# B&R Automation Studio project NAEUL004C00R13L518F00 (part 12)

#### Act_EntP0200Disp.st
```iecst
ACTION Act_EntP0200Disp:

	//Access Address
	p_tyC0005Main ACCESS ADR(tyCommon.tyMain);

	p_tyC0007Notif ACCESS ADR(tyCommon.tyNotif);

	p_tyC0008MsgBox ACCESS ADR(tyP0200OpsGen.tyMsgBoxHide);

	p_tyC0009Info ACCESS ADR(tyCommon.tyInfo);

	p_tyC0010RcyMsg ACCESS ADR(tyP0200OpsGen.tyRcyMsgHide);

	p_tyP0200OpsGen ACCESS ADR(tyP0200OpsGen.tyOps);
	p_tyP0200OpsOven ACCESS ADR(tyP0200OpsGen.tyOven);
	p_tyP0200OpsUSCommB ACCESS ADR(tyP0200OpsGen.tyUSCommB);
	p_tyP0200OpsUSAVSMEMA ACCESS ADR(tyP0200OpsGen.tyUSAVSMEMA);
	p_tyP0200OpsUSBVSMEMA ACCESS ADR(tyP0200OpsGen.tyUSBVSMEMA);
	p_tyP0200OpsUSAVSMEMA1 ACCESS ADR(tyP0200OpsGen.tyUSAVSMEMA1);
	p_tyP0200OpsUSBVSMEMA1 ACCESS ADR(tyP0200OpsGen.tyUSBVSMEMA1);
	p_tyP0200OpsBypsInitConv ACCESS ADR(tyP0200OpsGen.tyBypsInitConv);

	//Display
	tyP0200OpsGen.tyOven.tyLyr.uiRtStat.0	:= NOT(p_tyNtParamCurr.bOvenInfoPrep AND p_tyMcParamCurr.bOvenEn);

	//Communication - Upstream A
	IF p_tyMcParamCurr.eUSCommA = McSetCommModHermes THEN
		tyP0200OpsGen.tyOps.tyBitmapUSAComm.usiValueIdx	:= 1;
		tyP0200OpsGen.tyOps.tyBitmapUSAComm1.usiValueIdx	:= 1;

	ELSIF p_tyMcParamCurr.eUSCommA = McSetCommModSMEMA THEN
		tyP0200OpsGen.tyOps.tyBitmapUSAComm.usiValueIdx	:= 0;
		tyP0200OpsGen.tyOps.tyBitmapUSAComm1.usiValueIdx	:= 0;

	END_IF

	//Communication - Upstream B
	IF p_tyMcParamCurr.eUSCommB = McSetCommModHermes THEN
		tyP0200OpsGen.tyUSCommB.tyBitmapUSBComm.usiValueIdx	:= 1;
		tyP0200OpsGen.tyUSCommB.tyBitmapUSBComm1.usiValueIdx	:= 1;

	ELSIF p_tyMcParamCurr.eUSCommB = McSetCommModSMEMA THEN
		tyP0200OpsGen.tyUSCommB.tyBitmapUSBComm.usiValueIdx	:= 0;
		tyP0200OpsGen.tyUSCommB.tyBitmapUSBComm1.usiValueIdx	:= 0;

	END_IF

	//Virtual SMEMA
	IF (p_tyUsrMgmtCurrUsr.eUsrLvl = UsrMgmtLvl1) OR p_tyNtParamCurr.bVSMEMAPrep = FALSE OR p_tyMcParamCurr.bVSMEMAEn = FALSE OR (p_tyMcParamCurr.eUSCommA = McSetCommModHermes AND p_tyMcParamCurr.eUSCommB = McSetCommModHermes) THEN

		tyP0200OpsGen.tyOps.tyHotspotUSAVSMEMA.bValue		:= FALSE;
		tyP0200OpsGen.tyUSCommB.tyHotspotUSBVSMEMA.bValue	:= FALSE;
		tyP0200OpsGen.tyOps.tyHotspotUSAVSMEMA1.bValue		:= FALSE;
		tyP0200OpsGen.tyUSCommB.tyHotspotUSBVSMEMA1.bValue	:= FALSE;

		memset(ADR(tyP0200OpsGen.tyUSAVSMEMA), 0, SIZEOF(tyP0200OpsGen.tyUSAVSMEMA));
		memset(ADR(tyP0200OpsGen.tyUSBVSMEMA), 0, SIZEOF(tyP0200OpsGen.tyUSBVSMEMA));
		memset(ADR(tyP0200OpsGen.tyUSAVSMEMA1), 0, SIZEOF(tyP0200OpsGen.tyUSAVSMEMA1));
		memset(ADR(tyP0200OpsGen.tyUSBVSMEMA1), 0, SIZEOF(tyP0200OpsGen.tyUSBVSMEMA1));

		fUIInRtStatHide(ADR(tyP0200OpsGen.tyOps.tyHotspotUSAVSMEMA.uiRtStat));
		fUIInRtStatHide(ADR(tyP0200OpsGen.tyUSCommB.tyHotspotUSBVSMEMA.uiRtStat));
		fUIInRtStatHide(ADR(tyP0200OpsGen.tyUSAVSMEMA.tyLyr.uiRtStat));
		fUIInRtStatHide(ADR(tyP0200OpsGen.tyUSBVSMEMA.tyLyr.uiRtStat));

		fUIInRtStatHide(ADR(tyP0200OpsGen.tyOps.tyHotspotUSAVSMEMA1.uiRtStat));
		fUIInRtStatHide(ADR(tyP0200OpsGen.tyUSCommB.tyHotspotUSBVSMEMA1.uiRtStat));
		fUIInRtStatHide(ADR(tyP0200OpsGen.tyUSAVSMEMA1.tyLyr.uiRtStat));
		fUIInRtStatHide(ADR(tyP0200OpsGen.tyUSBVSMEMA1.tyLyr.uiRtStat));

		bVSMEMAUSAEn	:= FALSE;
		bVSMEMAUSBEn	:= FALSE;

	ELSE

		//Upstream A
		IF p_tyMcParamCurr.eUSCommA = McSetCommModHermes THEN
			tyP0200OpsGen.tyOps.tyHotspotUSAVSMEMA.bValue	:= FALSE;
			tyP0200OpsGen.tyOps.tyHotspotUSAVSMEMA1.bValue	:= FALSE;

			memset(ADR(tyP0200OpsGen.tyUSAVSMEMA), 0, SIZEOF(tyP0200OpsGen.tyUSAVSMEMA));

			fUIInRtStatHide(ADR(tyP0200OpsGen.tyOps.tyHotspotUSAVSMEMA.uiRtStat));
			fUIInRtStatHide(ADR(tyP0200OpsGen.tyUSAVSMEMA.tyLyr.uiRtStat));

			memset(ADR(tyP0200OpsGen.tyUSAVSMEMA1), 0, SIZEOF(tyP0200OpsGen.tyUSAVSMEMA1));

			fUIInRtStatHide(ADR(tyP0200OpsGen.tyOps.tyHotspotUSAVSMEMA1.uiRtStat));
			fUIInRtStatHide(ADR(tyP0200OpsGen.tyUSAVSMEMA1.tyLyr.uiRtStat));

		ELSIF p_tyMcParamCurr.eUSCommA = McSetCommModSMEMA THEN

			IF p_tyNtParamCurr.bUIConvDirRL = FALSE THEN
				tyP0200OpsGen.tyOps.tyHotspotUSAVSMEMA1.bValue	:= FALSE;
				fUIInRtStatHide(ADR(tyP0200OpsGen.tyUSAVSMEMA1.tyBtnStat.uiRtStat));
				fUIInRtStatHide(ADR(tyP0200OpsGen.tyUSAVSMEMA1.tyBtnDual.uiRtStat));
				fUIInRtStatHide(ADR(tyP0200OpsGen.tyUSAVSMEMA1.tyBtnNom.uiRtStat));

				memset(ADR(tyP0200OpsGen.tyUSAVSMEMA1), 0, SIZEOF(tyP0200OpsGen.tyUSAVSMEMA1));
				fUIInRtStatHide(ADR(tyP0200OpsGen.tyOps.tyHotspotUSAVSMEMA1.uiRtStat));
				fUIInRtStatHide(ADR(tyP0200OpsGen.tyUSAVSMEMA1.tyLyr.uiRtStat));

				fUIInRtStatOff(ADR(tyP0200OpsGen.tyOps.tyHotspotUSAVSMEMA.uiRtStat));
				fUIInRtStatOff(ADR(tyP0200OpsGen.tyOps.tyHotspotUSAVSMEMA1.uiRtStat));
				//Stat & Dual
				IF p_tyMcParamCurr.tyUSCommASMEMA.eSelection = SMEMASelIPC9851Ext THEN
					fUIInRtStatOff(ADR(tyP0200OpsGen.tyUSAVSMEMA.tyBtnStat.uiRtStat));
					fUIInRtStatOff(ADR(tyP0200OpsGen.tyUSAVSMEMA.tyBtnDual.uiRtStat));
				ELSE
					fUIInRtStatHide(ADR(tyP0200OpsGen.tyUSAVSMEMA.tyBtnStat.uiRtStat));
					fUIInRtStatHide(ADR(tyP0200OpsGen.tyUSAVSMEMA.tyBtnDual.uiRtStat));
				END_IF

			ELSE

				tyP0200OpsGen.tyOps.tyHotspotUSAVSMEMA.bValue	:= FALSE;
				fUIInRtStatHide(ADR(tyP0200OpsGen.tyUSAVSMEMA.tyBtnStat.uiRtStat));
				fUIInRtStatHide(ADR(tyP0200OpsGen.tyUSAVSMEMA.tyBtnDual.uiRtStat));
				fUIInRtStatHide(ADR(tyP0200OpsGen.tyUSAVSMEMA.tyBtnNom.uiRtStat));

				memset(ADR(tyP0200OpsGen.tyUSAVSMEMA), 0, SIZEOF(tyP0200OpsGen.tyUSAVSMEMA));
				fUIInRtStatHide(ADR(tyP0200OpsGen.tyOps.tyHotspotUSAVSMEMA.uiRtStat));
				fUIInRtStatHide(ADR(tyP0200OpsGen.tyUSAVSMEMA.tyLyr.uiRtStat));

				fUIInRtStatOff(ADR(tyP0200OpsGen.tyOps.tyHotspotUSAVSMEMA1.uiRtStat));

				//Stat & Dual
				IF p_tyMcParamCurr.tyUSCommASMEMA.eSelection = SMEMASelIPC9851Ext THEN
					fUIInRtStatOff(ADR(tyP0200OpsGen.tyUSAVSMEMA1.tyBtnStat.uiRtStat));
					fUIInRtStatOff(ADR(tyP0200OpsGen.tyUSAVSMEMA1.tyBtnDual.uiRtStat));
				ELSE
					fUIInRtStatHide(ADR(tyP0200OpsGen.tyUSAVSMEMA1.tyBtnStat.uiRtStat));
					fUIInRtStatHide(ADR(tyP0200OpsGen.tyUSAVSMEMA1.tyBtnDual.uiRtStat));
				END_IF

			END_IF

		END_IF

		//Upstream B
		IF p_tyNtParamCurr.bProjLaneBPrep THEN
			IF p_tyMcParamCurr.eUSCommB = McSetCommModHermes THEN
				tyP0200OpsGen.tyUSCommB.tyHotspotUSBVSMEMA.bValue	:= FALSE;
				tyP0200OpsGen.tyUSCommB.tyHotspotUSBVSMEMA1.bValue	:= FALSE;

				memset(ADR(tyP0200OpsGen.tyUSBVSMEMA), 0, SIZEOF(tyP0200OpsGen.tyUSBVSMEMA));

				fUIInRtStatHide(ADR(tyP0200OpsGen.tyUSCommB.tyHotspotUSBVSMEMA.uiRtStat));
				fUIInRtStatHide(ADR(tyP0200OpsGen.tyUSBVSMEMA.tyLyr.uiRtStat));

				memset(ADR(tyP0200OpsGen.tyUSBVSMEMA1), 0, SIZEOF(tyP0200OpsGen.tyUSBVSMEMA1));

				fUIInRtStatHide(ADR(tyP0200OpsGen.tyUSCommB.tyHotspotUSBVSMEMA1.uiRtStat));
				fUIInRtStatHide(ADR(tyP0200OpsGen.tyUSBVSMEMA1.tyLyr.uiRtStat));

			ELSIF p_tyMcParamCurr.eUSCommB = McSetCommModSMEMA THEN

				IF p_tyNtParamCurr.bUIConvDirRL = FALSE THEN
					tyP0200OpsGen.tyUSCommB.tyHotspotUSBVSMEMA1.bValue	:= FALSE;
					fUIInRtStatHide(ADR(tyP0200OpsGen.tyUSBVSMEMA1.tyBtnStat.uiRtStat));
					fUIInRtStatHide(ADR(tyP0200OpsGen.tyUSBVSMEMA1.tyBtnDual.uiRtStat));
					fUIInRtStatHide(ADR(tyP0200OpsGen.tyUSBVSMEMA1.tyBtnNom.uiRtStat));

					memset(ADR(tyP0200OpsGen.tyUSBVSMEMA1), 0, SIZEOF(tyP0200OpsGen.tyUSBVSMEMA1));
					fUIInRtStatHide(ADR(tyP0200OpsGen.tyUSCommB.tyHotspotUSBVSMEMA1.uiRtStat));
					fUIInRtStatHide(ADR(tyP0200OpsGen.tyUSBVSMEMA1.tyLyr.uiRtStat));

					fUIInRtStatOff(ADR(tyP0200OpsGen.tyUSCommB.tyHotspotUSBVSMEMA.uiRtStat));

					//Stat & Dual
					IF p_tyMcParamCurr.tyUSCommBSMEMA.eSelection = SMEMASelIPC9851Ext THEN
						fUIInRtStatOff(ADR(tyP0200OpsGen.tyUSBVSMEMA.tyBtnStat.uiRtStat));
						fUIInRtStatOff(ADR(tyP0200OpsGen.tyUSBVSMEMA.tyBtnDual.uiRtStat));
					ELSE
						fUIInRtStatHide(ADR(tyP0200OpsGen.tyUSBVSMEMA.tyBtnStat.uiRtStat));
						fUIInRtStatHide(ADR(tyP0200OpsGen.tyUSBVSMEMA.tyBtnDual.uiRtStat));
					END_IF

				ELSE
					tyP0200OpsGen.tyUSCommB.tyHotspotUSBVSMEMA.bValue	:= FALSE;
					fUIInRtStatHide(ADR(tyP0200OpsGen.tyUSBVSMEMA.tyBtnStat.uiRtStat));
					fUIInRtStatHide(ADR(tyP0200OpsGen.tyUSBVSMEMA.tyBtnDual.uiRtStat));
					fUIInRtStatHide(ADR(tyP0200OpsGen.tyUSBVSMEMA.tyBtnNom.uiRtStat));

					memset(ADR(tyP0200OpsGen.tyUSBVSMEMA), 0, SIZEOF(tyP0200OpsGen.tyUSBVSMEMA));
					fUIInRtStatHide(ADR(tyP0200OpsGen.tyUSCommB.tyHotspotUSBVSMEMA.uiRtStat));
					fUIInRtStatHide(ADR(tyP0200OpsGen.tyUSBVSMEMA.tyLyr.uiRtStat));

					fUIInRtStatOff(ADR(tyP0200OpsGen.tyUSCommB.tyHotspotUSBVSMEMA1.uiRtStat));

					//Stat & Dual
					IF p_tyMcParamCurr.tyUSCommBSMEMA.eSelection = SMEMASelIPC9851Ext THEN
						fUIInRtStatOff(ADR(tyP0200OpsGen.tyUSBVSMEMA1.tyBtnStat.uiRtStat));
						fUIInRtStatOff(ADR(tyP0200OpsGen.tyUSBVSMEMA1.tyBtnDual.uiRtStat));
					ELSE
						fUIInRtStatHide(ADR(tyP0200OpsGen.tyUSBVSMEMA1.tyBtnStat.uiRtStat));
						fUIInRtStatHide(ADR(tyP0200OpsGen.tyUSBVSMEMA1.tyBtnDual.uiRtStat));
					END_IF

				END_IF

			END_IF

		END_IF

	END_IF

	//General Operations Arrow Dislay

	IF p_tyNtParamCurr.bUIConvDirRL THEN

		tyP0200OpsGen.tyOps.tyBitmapDir1.usiValueIdx	:= 1;	// <<--
		tyP0200OpsGen.tyOps.tyBitmapDir2.usiValueIdx	:= 1;	// <<--
	ELSE

		tyP0200OpsGen.tyOps.tyBitmapDir1.usiValueIdx	:= 0;	// -->>
		tyP0200OpsGen.tyOps.tyBitmapDir2.usiValueIdx	:= 0;	// -->>

	END_IF

	//Disable AIV function
	IF p_tyNtParamCurr.bProjMagConvLane1Prep THEN
		fUIInRtStatHide(ADR(tyP0200OpsGen.tyOps.tyHotspotOpsAIV.uiMaskRtStat));
		IF p_tyMcParamCurr.bAGVComEn = FALSE THEN
			//			fUIInRtStatHide(ADR(tyP0200OpsGen.tyOps.tyHotspotOpsAIV.uiRtStat));
			fUIInRtStatOff(ADR(tyP0200OpsGen.tyOps.tyHotspotAIVGroup1Mask.uiMaskRtStat));
		ELSE
			//			fUIInRtStatOff(ADR(tyP0200OpsGen.tyOps.tyHotspotOpsAIV.uiRtStat));
			fUIInRtStatHide(ADR(tyP0200OpsGen.tyOps.tyHotspotAIVGroup1Mask.uiMaskRtStat));
		END_IF
	ELSE
		fUIInRtStatHide(ADR(tyP0200OpsGen.tyOps.tyHotspotAIVGroup1Mask.uiMaskRtStat));
		IF p_tyMcParamCurr.bAGVComEn = FALSE THEN
			//	fUIInRtStatHide(ADR(tyP0200OpsGen.tyOps.tyHotspotOpsAIV.uiRtStat));
			fUIInRtStatOff(ADR(tyP0200OpsGen.tyOps.tyHotspotOpsAIV.uiMaskRtStat));
		ELSE
			fUIInRtStatHide(ADR(tyP0200OpsGen.tyOps.tyHotspotOpsAIV.uiMaskRtStat));
		END_IF
	END_IF

	//AutoRcp
	IF NOT(p_bMcParamAutoRcpDisable) AND p_tyNtParamCurr.eAutoRcpPrecededBy =  PrecededBySelf THEN
		fUIInRtStatHide(ADR(tyP0200OpsGen.tyOps.tyNumPitch.uiRtStat));
		fUIInRtStatHide(ADR(tyP0200OpsGen.tyOps.tyNumMinSltRange.uiRtStat));
		fUIInRtStatHide(ADR(tyP0200OpsGen.tyOps.tyNumMaxSltRange.uiRtStat));
		fUIInRtStatHide(ADR(tyP0200OpsGen.tyOps.tyNumPitchRToL.uiRtStat));
		fUIInRtStatHide(ADR(tyP0200OpsGen.tyOps.tyNumMinSltRangeRToL.uiRtStat));
		fUIInRtStatHide(ADR(tyP0200OpsGen.tyOps.tyNumMaxSltRangeRToL.uiRtStat));
	ELSE  //PrecededByF1 OR p_bMcParamAutoRcpDisable
		tyP0200OpsGen.tyOps.tyNumPitch.uiRtStat.0 :=  p_tyNtParamCurr.bUIConvDirRL;
		tyP0200OpsGen.tyOps.tyNumMinSltRange.uiRtStat.0 := p_tyNtParamCurr.bUIConvDirRL;
		tyP0200OpsGen.tyOps.tyNumMaxSltRange.uiRtStat.0 := p_tyNtParamCurr.bUIConvDirRL;
		tyP0200OpsGen.tyOps.tyNumPitchRToL.uiRtStat.0 :=  NOT(p_tyNtParamCurr.bUIConvDirRL);
		tyP0200OpsGen.tyOps.tyNumMinSltRangeRToL.uiRtStat.0 := NOT(p_tyNtParamCurr.bUIConvDirRL);
		tyP0200OpsGen.tyOps.tyNumMaxSltRangeRToL.uiRtStat.0 := NOT(p_tyNtParamCurr.bUIConvDirRL);
	END_IF

END_ACTION
```

#### Act_OptP0200ChgPage.st
```iecst
ACTION Act_OptP0200ChgPage:

	IF tyP0200OpsGen.tyOps.tyHotspotOpsTravLifter.bRtCompl = TRUE THEN
		tyP0200OpsGen.tyOps.tyHotspotOpsTravLifter.bRtCompl	:= FALSE;

		eChgPage	:= UIP0201OpsTravLifter;

	ELSIF tyP0200OpsGen.tyOps.tyHotspotOps2Mag1.bRtCompl = TRUE OR tyP0200OpsGen.tyOps.tyHotspotOps3Mag1.bRtCompl = TRUE THEN
		tyP0200OpsGen.tyOps.tyHotspotOps2Mag1.bRtCompl	:= FALSE;
		tyP0200OpsGen.tyOps.tyHotspotOps3Mag1.bRtCompl	:= FALSE;

		eChgPage	:= UIP0202OpsMag1;

	ELSIF tyP0200OpsGen.tyOps.tyHotspotOps2Mag2.bRtCompl = TRUE OR tyP0200OpsGen.tyOps.tyHotspotOps3Mag2.bRtCompl = TRUE THEN
		tyP0200OpsGen.tyOps.tyHotspotOps2Mag2.bRtCompl	:= FALSE;
		tyP0200OpsGen.tyOps.tyHotspotOps3Mag2.bRtCompl	:= FALSE;

		eChgPage	:= UIP0203OpsMag2;

	ELSIF tyP0200OpsGen.tyOps.tyHotspotOps3Mag3.bRtCompl = TRUE THEN
		tyP0200OpsGen.tyOps.tyHotspotOps3Mag3.bRtCompl	:= FALSE;

		eChgPage	:= UIP0204OpsMag3;

	ELSIF tyP0200OpsGen.tyOps.tyHotspotOpsAIV.bRtCompl = TRUE THEN
		tyP0200OpsGen.tyOps.tyHotspotOpsAIV.bRtCompl	:= FALSE;

		eChgPage	:= UIP0205OpsAIV;

	ELSIF tyP0200OpsGen.tyOps.tyHotspotOpsMagLane1.bRtCompl = TRUE THEN
		tyP0200OpsGen.tyOps.tyHotspotOpsMagLane1.bRtCompl	:= FALSE;

		eChgPage	:= UIP0206OpsMagConv1;

	ELSIF tyP0200OpsGen.tyOps.tyHotspotOpsMagLane2.bRtCompl = TRUE THEN
		tyP0200OpsGen.tyOps.tyHotspotOpsMagLane2.bRtCompl	:= FALSE;

		eChgPage	:= UIP0207OpsMagConv2;

	ELSIF tyP0200OpsGen.tyOps.tyHotspotOpsMagInfo.bRtCompl = TRUE THEN
		tyP0200OpsGen.tyOps.tyHotspotOpsMagInfo.bRtCompl	:= FALSE;

		eChgPage	:= UIP0800MagInfo;

	ELSIF tyP0200OpsGen.tyOven.tyHotspotOven.bRtCompl = TRUE THEN
		tyP0200OpsGen.tyOven.tyHotspotOven.bRtCompl	:= FALSE;

		eChgPage	:= UIP0850OvenInfo;

	END_IF

END_ACTION
```

#### Act_OptP0200UpdtDat.st
```iecst
ACTION Act_OptP0200UpdtDat:

	//PCB Status
	IF p_bPshrConvHvBrd = TRUE THEN
		IF p_bPshrConvGdBrd = TRUE THEN
			tyP0200OpsGen.tyOps.tyBitmapPCB.usiValueIdx	:= 1;
		ELSE
			tyP0200OpsGen.tyOps.tyBitmapPCB.usiValueIdx	:= 2;
		END_IF
	ELSE
		tyP0200OpsGen.tyOps.tyBitmapPCB.usiValueIdx	:= 0;
	END_IF

	//Communication - Mask
	IF p_tyNtParamCurr.bUIConvDirRL = FALSE THEN
		fUIInRtStatHide(ADR(tyP0200OpsGen.tyOps.tyBitmapUSAComm1.uiMaskRtStat));
		fUIInRtStatHide(ADR(tyP0200OpsGen.tyUSCommB.tyBitmapUSBComm1.uiMaskRtStat));
		IF p_tyMcParamCurr.eUSCommA = McSetCommModSMEMA THEN
			fUIInRtStatHide(ADR(tyP0200OpsGen.tyOps.tyBitmapUSAComm.uiMaskRtStat));
		ELSIF p_tyMcParamCurr.eUSCommA = McSetCommModHermes THEN
			IF p_bUSHermesAConnected = TRUE THEN
				fUIInRtStatHide(ADR(tyP0200OpsGen.tyOps.tyBitmapUSAComm.uiMaskRtStat));
			ELSE
				fUIInRtStatOff(ADR(tyP0200OpsGen.tyOps.tyBitmapUSAComm.uiMaskRtStat));
			END_IF
		END_IF

		IF p_tyMcParamCurr.eUSCommB = McSetCommModSMEMA THEN
			fUIInRtStatHide(ADR(tyP0200OpsGen.tyUSCommB.tyBitmapUSBComm.uiMaskRtStat));
		ELSIF p_tyMcParamCurr.eUSCommB = McSetCommModHermes THEN
			IF p_bUSHermesBConnected = TRUE THEN
				fUIInRtStatHide(ADR(tyP0200OpsGen.tyUSCommB.tyBitmapUSBComm.uiMaskRtStat));
			ELSE
				fUIInRtStatOff(ADR(tyP0200OpsGen.tyUSCommB.tyBitmapUSBComm.uiMaskRtStat));
			END_IF
		END_IF
	ELSE
		fUIInRtStatHide(ADR(tyP0200OpsGen.tyOps.tyBitmapUSAComm.uiMaskRtStat));
		fUIInRtStatHide(ADR(tyP0200OpsGen.tyUSCommB.tyBitmapUSBComm.uiMaskRtStat));
		IF p_tyMcParamCurr.eUSCommA = McSetCommModSMEMA THEN
			fUIInRtStatHide(ADR(tyP0200OpsGen.tyOps.tyBitmapUSAComm1.uiMaskRtStat));
		ELSIF p_tyMcParamCurr.eUSCommA = McSetCommModHermes THEN
			IF p_bUSHermesAConnected = TRUE THEN
				fUIInRtStatHide(ADR(tyP0200OpsGen.tyOps.tyBitmapUSAComm1.uiMaskRtStat));
			ELSE
				fUIInRtStatOff(ADR(tyP0200OpsGen.tyOps.tyBitmapUSAComm1.uiMaskRtStat));
			END_IF
		END_IF

		IF p_tyMcParamCurr.eUSCommB = McSetCommModSMEMA THEN
			fUIInRtStatHide(ADR(tyP0200OpsGen.tyUSCommB.tyBitmapUSBComm1.uiMaskRtStat));
		ELSIF p_tyMcParamCurr.eUSCommB = McSetCommModHermes THEN
			IF p_bUSHermesBConnected = TRUE THEN
				fUIInRtStatHide(ADR(tyP0200OpsGen.tyUSCommB.tyBitmapUSBComm1.uiMaskRtStat));
			ELSE
				fUIInRtStatOff(ADR(tyP0200OpsGen.tyUSCommB.tyBitmapUSBComm1.uiMaskRtStat));
			END_IF
		END_IF
	END_IF
	//Communication - Signal
	//USB A
	IF p_tyMcParamCurr.eUSCommA = McSetCommModSMEMA THEN
		IF p_tyNtParamCurr.bUIConvDirRL = FALSE THEN

			IF p_bUSSMEMAADSRdy = TRUE THEN
				tyP0200OpsGen.tyOps.tyBitmapUSOut.usiValueIdx	:= 1;
			ELSE
				tyP0200OpsGen.tyOps.tyBitmapUSOut.usiValueIdx	:= 0;
			END_IF
		ELSE
			IF p_bUSSMEMAADSRdy = TRUE THEN
				tyP0200OpsGen.tyOps.tyBitmapUSOut1.usiValueIdx	:= 1;
			ELSE
				tyP0200OpsGen.tyOps.tyBitmapUSOut1.usiValueIdx	:= 0;
			END_IF
		END_IF

	ELSIF p_tyMcParamCurr.eUSCommA = McSetCommModHermes THEN
		IF p_tyNtParamCurr.bUIConvDirRL = FALSE THEN
			IF p_bUSHermesADSRdy = TRUE THEN
				IF p_bUSHermesADSGdRdy = TRUE THEN
					tyP0200OpsGen.tyOps.tyBitmapUSOut.usiValueIdx	:= 1;
				ELSE
					tyP0200OpsGen.tyOps.tyBitmapUSOut.usiValueIdx	:= 2;
				END_IF
			ELSE
				tyP0200OpsGen.tyOps.tyBitmapUSOut.usiValueIdx		:= 0;
			END_IF
		ELSE
			IF p_bUSHermesADSRdy = TRUE THEN
				IF p_bUSHermesADSGdRdy = TRUE THEN
					tyP0200OpsGen.tyOps.tyBitmapUSOut1.usiValueIdx	:= 1;
				ELSE
					tyP0200OpsGen.tyOps.tyBitmapUSOut1.usiValueIdx	:= 2;
				END_IF
			ELSE
				tyP0200OpsGen.tyOps.tyBitmapUSOut1.usiValueIdx		:= 0;
			END_IF
		END_IF

	END_IF

	//UBA A
	IF p_tyMcParamCurr.eUSCommA = McSetCommModSMEMA THEN

	IF p_tyNtParamCurr.bUIConvDirRL = FALSE THEN
		IF p_bUSSMEMAAUSRdy = TRUE THEN
			IF p_bUSSMEMAAUSGdBrdRdy = TRUE THEN
				tyP0200OpsGen.tyOps.tyBitmapUSIn.usiValueIdx	:= 1;
			ELSE
				tyP0200OpsGen.tyOps.tyBitmapUSIn.usiValueIdx	:= 2;
			END_IF
		ELSE
			tyP0200OpsGen.tyOps.tyBitmapUSIn.usiValueIdx		:= 0;
		END_IF
	ELSE
		IF p_bUSSMEMAAUSRdy = TRUE THEN
			IF p_bUSSMEMAAUSGdBrdRdy = TRUE THEN
				tyP0200OpsGen.tyOps.tyBitmapUSIn1.usiValueIdx	:= 1;
			ELSE
				tyP0200OpsGen.tyOps.tyBitmapUSIn1.usiValueIdx	:= 2;
			END_IF
		ELSE
			tyP0200OpsGen.tyOps.tyBitmapUSIn1.usiValueIdx		:= 0;
		END_IF
	END_IF

	ELSIF p_tyMcParamCurr.eUSCommA = McSetCommModHermes THEN

		IF p_tyNtParamCurr.bUIConvDirRL = FALSE THEN
			IF p_bUSHermesAUSRdy = TRUE THEN
				IF p_bUSHermesAUSGdRdy = TRUE THEN
					tyP0200OpsGen.tyOps.tyBitmapUSIn.usiValueIdx	:= 1;
				ELSE
					tyP0200OpsGen.tyOps.tyBitmapUSIn.usiValueIdx	:= 2;
				END_IF
			ELSE
				tyP0200OpsGen.tyOps.tyBitmapUSIn.usiValueIdx		:= 0;
			END_IF
		ELSE
			IF p_bUSHermesAUSRdy = TRUE THEN
				IF p_bUSHermesAUSGdRdy = TRUE THEN
					tyP0200OpsGen.tyOps.tyBitmapUSIn1.usiValueIdx	:= 1;
				ELSE
					tyP0200OpsGen.tyOps.tyBitmapUSIn1.usiValueIdx	:= 2;
				END_IF
			ELSE
				tyP0200OpsGen.tyOps.tyBitmapUSIn1.usiValueIdx		:= 0;
			END_IF
		END_IF

	END_IF

	//USB B
	IF p_tyMcParamCurr.eUSCommB = McSetCommModSMEMA THEN
		IF p_tyNtParamCurr.bUIConvDirRL = FALSE THEN

			IF p_bUSSMEMABDSRdy = TRUE THEN
				tyP0200OpsGen.tyUSCommB.tyBitmapUSOut.usiValueIdx	:= 1;
			ELSE
				tyP0200OpsGen.tyUSCommB.tyBitmapUSOut.usiValueIdx	:= 0;
			END_IF

		ELSE

			IF p_bUSSMEMABDSRdy = TRUE THEN
				tyP0200OpsGen.tyUSCommB.tyBitmapUSOut1.usiValueIdx	:= 1;
			ELSE
				tyP0200OpsGen.tyUSCommB.tyBitmapUSOut1.usiValueIdx	:= 0;
			END_IF

		END_IF

	ELSIF p_tyMcParamCurr.eUSCommB = McSetCommModHermes THEN

		IF p_tyNtParamCurr.bUIConvDirRL THEN
			IF p_bUSHermesBDSRdy = TRUE THEN
				IF p_bUSHermesBDSGdRdy = TRUE THEN
					tyP0200OpsGen.tyUSCommB.tyBitmapUSOut.usiValueIdx	:= 1;
				ELSE
					tyP0200OpsGen.tyUSCommB.tyBitmapUSOut.usiValueIdx	:= 2;
				END_IF
			ELSE
				tyP0200OpsGen.tyUSCommB.tyBitmapUSOut.usiValueIdx		:= 0;
			END_IF
		ELSE
			IF p_bUSHermesBDSRdy = TRUE THEN
				IF p_bUSHermesBDSGdRdy = TRUE THEN
					tyP0200OpsGen.tyUSCommB.tyBitmapUSOut1.usiValueIdx	:= 1;
				ELSE
					tyP0200OpsGen.tyUSCommB.tyBitmapUSOut1.usiValueIdx	:= 2;
				END_IF
			ELSE
				tyP0200OpsGen.tyUSCommB.tyBitmapUSOut1.usiValueIdx		:= 0;
			END_IF
		END_IF

	END_IF

	//UBA B
	IF p_tyMcParamCurr.eUSCommB = McSetCommModSMEMA THEN

		IF p_tyNtParamCurr.bUIConvDirRL = FALSE THEN
			IF p_bUSSMEMABUSRdy = TRUE THEN
				IF p_bUSSMEMABUSGdBrdRdy = TRUE THEN
					tyP0200OpsGen.tyUSCommB.tyBitmapUSIn.usiValueIdx	:= 1;
				ELSE
					tyP0200OpsGen.tyUSCommB.tyBitmapUSIn.usiValueIdx	:= 2;
				END_IF
			ELSE
				tyP0200OpsGen.tyUSCommB.tyBitmapUSIn.usiValueIdx		:= 0;
			END_IF
		ELSE
			IF p_bUSSMEMABUSRdy = TRUE THEN
				IF p_bUSSMEMABUSGdBrdRdy = TRUE THEN
					tyP0200OpsGen.tyUSCommB.tyBitmapUSIn1.usiValueIdx	:= 1;
				ELSE
					tyP0200OpsGen.tyUSCommB.tyBitmapUSIn1.usiValueIdx	:= 2;
				END_IF
			ELSE
				tyP0200OpsGen.tyUSCommB.tyBitmapUSIn1.usiValueIdx		:= 0;
			END_IF
		END_IF

	ELSIF p_tyMcParamCurr.eUSCommB = McSetCommModHermes THEN

		IF p_tyNtParamCurr.bUIConvDirRL = FALSE THEN
			IF p_bUSHermesBUSRdy = TRUE THEN
				IF p_bUSHermesBUSGdRdy = TRUE THEN
					tyP0200OpsGen.tyUSCommB.tyBitmapUSIn.usiValueIdx	:= 1;
				ELSE
					tyP0200OpsGen.tyUSCommB.tyBitmapUSIn.usiValueIdx	:= 2;
				END_IF
			ELSE
				tyP0200OpsGen.tyUSCommB.tyBitmapUSIn.usiValueIdx		:= 0;
			END_IF
		ELSE
			IF p_bUSHermesBUSRdy = TRUE THEN
				IF p_bUSHermesBUSGdRdy = TRUE THEN
					tyP0200OpsGen.tyUSCommB.tyBitmapUSIn1.usiValueIdx	:= 1;
				ELSE
					tyP0200OpsGen.tyUSCommB.tyBitmapUSIn1.usiValueIdx	:= 2;
				END_IF
			ELSE
				tyP0200OpsGen.tyUSCommB.tyBitmapUSIn1.usiValueIdx		:= 0;
			END_IF
		END_IF

	END_IF

	//Alarm
	IF NOT p_bAlarmErr THEN
		memset(ADR(tyUIAlmData.bAlm) , 0 , SIZEOF(tyUIAlmData.bAlm));
	END_IF

	IF NOT p_bAlarmWarning THEN
		memset(ADR(tyUIAlmData.bWarning) , 0 , SIZEOF(tyUIAlmData.bWarning));
	ELSE
		IF p_bUSHermesAConnected OR p_tyMcParamCurr.eUSCommA = McSetCommModSMEMA THEN
			tyUIAlmData.bWarning[3114] := FALSE;
		END_IF
		IF p_bUSHermesBConnected OR p_tyMcParamCurr.eUSCommB = McSetCommModSMEMA THEN
			tyUIAlmData.bWarning[3281] := FALSE;
		END_IF
	END_IF

	FOR i := 1 TO c_uiP0200TableSize DO
		IF p_bStartupUISettingsLoadDone THEN
			IF p_tyAlarmCurrList[i].eSeverity = AlmSeverityError THEN
				tyUIAlmData.bAlm[p_tyAlarmCurrList[i].udiErrorCode] := p_tyAlarmCurrList[i].bAlm;
			ELSIF p_tyAlarmCurrList[i].eSeverity = AlmSeverityWarning THEN
				tyUIAlmData.bWarning[p_tyAlarmCurrList[i].udiErrorCode] := p_tyAlarmCurrList[i].bWarning;
			END_IF
		END_IF
	END_FOR

	//Magazine Info
	IF NOT(p_tyNtParamCurr.bAutoRcpPrep) OR  ( p_tyNtParamCurr.bAutoRcpPrep AND  p_bMcParamAutoRcpDisable) THEN
		tyP0200OpsGen.tyOps.tyNumMinSltRange.diValue	:= p_tyProdRcpCurrRcp2.diMinSltValue;
		tyP0200OpsGen.tyOps.tyNumMaxSltRange.diValue	:= p_tyProdRcpCurrRcp2.diMaxSltValue;
		tyP0200OpsGen.tyOps.tyNumPitch.diValue			:= p_tyProdRcpCurrRcp2.diPitch;
	ELSIF p_tyNtParamCurr.eAutoRcpPrecededBy =  PrecededByF1 THEN
		tyP0200OpsGen.tyOps.tyNumMinSltRange.diValue	:= p_tyProdRcpCurrRcp1.diMinSltValue; //update immediately based on LCS Running Rcp
		tyP0200OpsGen.tyOps.tyNumMaxSltRange.diValue	:= p_tyProdRcpCurrRcp1.diMaxSltValue;
		tyP0200OpsGen.tyOps.tyNumPitch.diValue			:= p_tyProdRcpCurrRcp1.diPitch;
	END_IF

	//Mag1
	IF p_bBuffer1MagPresent = TRUE THEN
		IF (p_tyNtParamCurr.eCustomerReq = Siemens OR p_tyNtParamCurr.eCustomerReq = We_Fabricate)AND p_iOpsMagConvUL1MESAcptCond <= 0 AND p_tyMcParamCurr.bMESEn THEN
			tyP0200OpsGen.tyOps.tyNumMag1AvlQty.diValue	:= 0;
			tyP0200OpsGen.tyOps.tyNumMag1TtlSlt.diValue	:= 0;
		ELSE
			tyP0200OpsGen.tyOps.tyNumMag1AvlQty.diValue		:= p_tyBuffer1BffrStat.diTtlBrdCap - (p_tyBuffer1BffrStat.diTtlBadBrd + p_tyBuffer1BffrStat.diTtlGdBrd);
			tyP0200OpsGen.tyOps.tyNumMag1TtlSlt.diValue		:= p_tyBuffer1BffrStat.diTtlBrdCap;
		END_IF
	ELSE
		tyP0200OpsGen.tyOps.tyNumMag1AvlQty.diValue		:= 0;
		tyP0200OpsGen.tyOps.tyNumMag1TtlSlt.diValue		:= 0;
	END_IF

	//Mag2
	IF p_bBuffer2MagPresent = TRUE THEN
		IF (p_tyNtParamCurr.eCustomerReq = Siemens OR p_tyNtParamCurr.eCustomerReq = We_Fabricate) AND p_iOpsMagConvUL2MESAcptCond <= 0 AND p_tyMcParamCurr.bMESEn THEN
			tyP0200OpsGen.tyOps.tyNumMag2AvlQty.diValue	:= 0;
			tyP0200OpsGen.tyOps.tyNumMag2TtlSlt.diValue		:= 0;
		ELSE
			tyP0200OpsGen.tyOps.tyNumMag2AvlQty.diValue		:= p_tyBuffer2BffrStat.diTtlBrdCap - (p_tyBuffer2BffrStat.diTtlBadBrd + p_tyBuffer2BffrStat.diTtlGdBrd);
			tyP0200OpsGen.tyOps.tyNumMag2TtlSlt.diValue		:= p_tyBuffer2BffrStat.diTtlBrdCap;
		END_IF
	ELSE
		tyP0200OpsGen.tyOps.tyNumMag2AvlQty.diValue		:= 0;
		tyP0200OpsGen.tyOps.tyNumMag2TtlSlt.diValue		:= 0;
	END_IF
	//Mag3
	IF p_bBuffer3MagPresent = TRUE THEN
		IF (p_tyNtParamCurr.eCustomerReq = Siemens OR p_tyNtParamCurr.eCustomerReq = We_Fabricate) AND p_iOpsMagConvUL3MESAcptCond <= 0 AND  p_tyMcParamCurr.bMESEn THEN
			tyP0200OpsGen.tyOps.tyNumMag3AvlQty.diValue		:= 0;
			tyP0200OpsGen.tyOps.tyNumMag3TtlSlt.diValue		:= 0;
		ELSE
			tyP0200OpsGen.tyOps.tyNumMag3AvlQty.diValue		:= p_tyBuffer3BffrStat.diTtlBrdCap - (p_tyBuffer3BffrStat.diTtlBadBrd + p_tyBuffer3BffrStat.diTtlGdBrd);
			tyP0200OpsGen.tyOps.tyNumMag3TtlSlt.diValue		:= p_tyBuffer3BffrStat.diTtlBrdCap;
		END_IF
	ELSE
		tyP0200OpsGen.tyOps.tyNumMag3AvlQty.diValue		:= 0;
		tyP0200OpsGen.tyOps.tyNumMag3TtlSlt.diValue		:= 0;
	END_IF

	//Oven
	tyP0200OpsGen.tyOven.tyBtnCntrA.bValue				:= p_tyDI.bOvenInfeedSigA;
	tyP0200OpsGen.tyOven.tyBtnCntrB.bValue				:= p_tyDI.bOvenInfeedSigB;
	tyP0200OpsGen.tyOven.tyBtnOvenA.bValue				:= p_tyDO.bOvenInfoSigA;
	tyP0200OpsGen.tyOven.tyBtnOvenB.bValue				:= p_tyDO.bOvenInfoSigB;

	//AIV TCP Bitmap
	IF p_tyNtParamCurr.bProjTCPAGVSigPrep THEN
		tyP0200OpsGen.tyOps.tyBitmapAIVTCP.usiValueIdx := BOOL_TO_USINT (p_bTCPConnected);
	END_IF
END_ACTION
```

#### Act_OptP0200VirtualSMEMA.st
```iecst
ACTION Act_OptP0200VSMEMA:

	//Upstream Virtual SMEMA A
	//Enable / Disable
	IF p_tyNtParamCurr.bUIConvDirRL = FALSE THEN
		IF tyP0200OpsGen.tyOps.tyHotspotUSAVSMEMA.bRtCompl = TRUE THEN
			tyP0200OpsGen.tyOps.tyHotspotUSAVSMEMA.bRtCompl	:= FALSE;

			IF tyP0200OpsGen.tyOps.tyHotspotUSAVSMEMA.bValue = TRUE THEN
				bVSMEMAUSAEn	:= TRUE;

				fUIInRtStatOff(ADR(tyP0200OpsGen.tyUSAVSMEMA.tyLyr.uiRtStat));
				fUIInRtStatHide(ADR(tyP0200OpsGen.tyUSAVSMEMA1.tyLyr.uiRtStat));
			ELSE
				tyP0200OpsGen.tyUSAVSMEMA.tyBtnNom.bValue	:= FALSE;
				tyP0200OpsGen.tyUSAVSMEMA.tyBtnStat.bValue	:= FALSE;
				tyP0200OpsGen.tyUSAVSMEMA.tyBtnDual.bValue	:= FALSE;

				bVSMEMAUSAEn	:= FALSE;

				fUIInRtStatHide(ADR(tyP0200OpsGen.tyUSAVSMEMA.tyLyr.uiRtStat));
				fUIInRtStatHide(ADR(tyP0200OpsGen.tyUSAVSMEMA1.tyLyr.uiRtStat));
			END_IF

		END_IF
	ELSE
		IF tyP0200OpsGen.tyOps.tyHotspotUSAVSMEMA1.bRtCompl = TRUE THEN
			tyP0200OpsGen.tyOps.tyHotspotUSAVSMEMA1.bRtCompl	:= FALSE;

			IF tyP0200OpsGen.tyOps.tyHotspotUSAVSMEMA1.bValue = TRUE THEN
				bVSMEMAUSAEn	:= TRUE;

				fUIInRtStatOff(ADR(tyP0200OpsGen.tyUSAVSMEMA1.tyLyr.uiRtStat));
				fUIInRtStatHide(ADR(tyP0200OpsGen.tyUSAVSMEMA.tyLyr.uiRtStat));
			ELSE
				tyP0200OpsGen.tyUSAVSMEMA.tyBtnNom.bValue	:= FALSE;
				tyP0200OpsGen.tyUSAVSMEMA.tyBtnStat.bValue	:= FALSE;
				tyP0200OpsGen.tyUSAVSMEMA.tyBtnDual.bValue	:= FALSE;

				bVSMEMAUSAEn	:= FALSE;

				fUIInRtStatHide(ADR(tyP0200OpsGen.tyUSAVSMEMA.tyLyr.uiRtStat));
				fUIInRtStatHide(ADR(tyP0200OpsGen.tyUSAVSMEMA1.tyLyr.uiRtStat));
			END_IF

		END_IF

	END_IF

	//Control

	IF p_tyNtParamCurr.bUIConvDirRL = FALSE THEN
		IF tyP0200OpsGen.tyUSAVSMEMA.tyBtnDual.bRtCompl = TRUE THEN
			tyP0200OpsGen.tyUSAVSMEMA.tyBtnDual.bRtCompl	:= FALSE;

			IF tyP0200OpsGen.tyUSAVSMEMA.tyBtnDual.bValue = TRUE THEN
				tyP0200OpsGen.tyUSAVSMEMA.tyBtnNom.bValue	:= TRUE;
				tyP0200OpsGen.tyUSAVSMEMA.tyBtnStat.bValue	:= TRUE;
			ELSE
				tyP0200OpsGen.tyUSAVSMEMA.tyBtnNom.bValue	:= FALSE;
				tyP0200OpsGen.tyUSAVSMEMA.tyBtnStat.bValue	:= FALSE;
			END_IF

		ELSIF tyP0200OpsGen.tyUSAVSMEMA.tyBtnNom.bRtCompl = TRUE THEN
			tyP0200OpsGen.tyUSAVSMEMA.tyBtnNom.bRtCompl	:= FALSE;

			IF tyP0200OpsGen.tyUSAVSMEMA.tyBtnNom.bValue = TRUE THEN
				IF tyP0200OpsGen.tyUSAVSMEMA.tyBtnStat.bValue =  TRUE THEN
					tyP0200OpsGen.tyUSAVSMEMA.tyBtnDual.bValue	:= TRUE;
				END_IF
			ELSE
				tyP0200OpsGen.tyUSAVSMEMA.tyBtnDual.bValue	:= FALSE;
			END_IF

		ELSIF tyP0200OpsGen.tyUSAVSMEMA.tyBtnStat.bRtCompl = TRUE THEN
			tyP0200OpsGen.tyUSAVSMEMA.tyBtnStat.bRtCompl	:= FALSE;

			IF tyP0200OpsGen.tyUSAVSMEMA.tyBtnStat.bValue = TRUE THEN
				IF tyP0200OpsGen.tyUSAVSMEMA.tyBtnNom.bValue =  TRUE THEN
					tyP0200OpsGen.tyUSAVSMEMA.tyBtnDual.bValue	:= TRUE;
				END_IF
			ELSE
				tyP0200OpsGen.tyUSAVSMEMA.tyBtnDual.bValue	:= FALSE;
			END_IF

		END_IF
	ELSE
		IF tyP0200OpsGen.tyUSAVSMEMA1.tyBtnDual.bRtCompl = TRUE THEN
			tyP0200OpsGen.tyUSAVSMEMA1.tyBtnDual.bRtCompl	:= FALSE;

			IF tyP0200OpsGen.tyUSAVSMEMA1.tyBtnDual.bValue = TRUE THEN
				tyP0200OpsGen.tyUSAVSMEMA1.tyBtnNom.bValue	:= TRUE;
				tyP0200OpsGen.tyUSAVSMEMA1.tyBtnStat.bValue	:= TRUE;
			ELSE
				tyP0200OpsGen.tyUSAVSMEMA1.tyBtnNom.bValue	:= FALSE;
				tyP0200OpsGen.tyUSAVSMEMA1.tyBtnStat.bValue	:= FALSE;
			END_IF

		ELSIF tyP0200OpsGen.tyUSAVSMEMA1.tyBtnNom.bRtCompl = TRUE THEN
			tyP0200OpsGen.tyUSAVSMEMA1.tyBtnNom.bRtCompl	:= FALSE;

			IF tyP0200OpsGen.tyUSAVSMEMA1.tyBtnNom.bValue = TRUE THEN
				IF tyP0200OpsGen.tyUSAVSMEMA1.tyBtnStat.bValue =  TRUE THEN
					tyP0200OpsGen.tyUSAVSMEMA1.tyBtnDual.bValue	:= TRUE;
				END_IF
			ELSE
				tyP0200OpsGen.tyUSAVSMEMA1.tyBtnDual.bValue	:= FALSE;
			END_IF

		ELSIF tyP0200OpsGen.tyUSAVSMEMA1.tyBtnStat.bRtCompl = TRUE THEN
			tyP0200OpsGen.tyUSAVSMEMA1.tyBtnStat.bRtCompl	:= FALSE;

			IF tyP0200OpsGen.tyUSAVSMEMA1.tyBtnStat.bValue = TRUE THEN
				IF tyP0200OpsGen.tyUSAVSMEMA1.tyBtnNom.bValue =  TRUE THEN
					tyP0200OpsGen.tyUSAVSMEMA1.tyBtnDual.bValue	:= TRUE;
				END_IF
			ELSE
				tyP0200OpsGen.tyUSAVSMEMA1.tyBtnDual.bValue	:= FALSE;
			END_IF

		END_IF
	END_IF

	//Update
	IF p_tyNtParamCurr.bUIConvDirRL = FALSE THEN
		bVSMEMAUBAA		:= tyP0200OpsGen.tyUSAVSMEMA.tyBtnNom.bValue;
		bVSMEMAUBAAStat	:= tyP0200OpsGen.tyUSAVSMEMA.tyBtnStat.bValue;
	ELSE
		bVSMEMAUBAA		:= tyP0200OpsGen.tyUSAVSMEMA1.tyBtnNom.bValue;
		bVSMEMAUBAAStat	:= tyP0200OpsGen.tyUSAVSMEMA1.tyBtnStat.bValue;
	END_IF

	//Upstream Virtual SMEMA B
	//Enable / Disable
	IF p_tyNtParamCurr.bUIConvDirRL = FALSE THEN
		IF tyP0200OpsGen.tyUSCommB.tyHotspotUSBVSMEMA.bRtCompl = TRUE THEN
			tyP0200OpsGen.tyUSCommB.tyHotspotUSBVSMEMA.bRtCompl	:= FALSE;

			IF tyP0200OpsGen.tyUSCommB.tyHotspotUSBVSMEMA.bValue = TRUE THEN
				bVSMEMAUSBEn	:= TRUE;

				fUIInRtStatOff(ADR(tyP0200OpsGen.tyUSBVSMEMA.tyLyr.uiRtStat));
				fUIInRtStatHide(ADR(tyP0200OpsGen.tyUSBVSMEMA1.tyLyr.uiRtStat));
			ELSE
				tyP0200OpsGen.tyUSBVSMEMA.tyBtnNom.bValue	:= FALSE;
				tyP0200OpsGen.tyUSBVSMEMA.tyBtnStat.bValue	:= FALSE;
				tyP0200OpsGen.tyUSBVSMEMA.tyBtnDual.bValue	:= FALSE;

				bVSMEMAUSBEn	:= FALSE;

				fUIInRtStatHide(ADR(tyP0200OpsGen.tyUSBVSMEMA.tyLyr.uiRtStat));
				fUIInRtStatHide(ADR(tyP0200OpsGen.tyUSBVSMEMA1.tyLyr.uiRtStat));
			END_IF

		END_IF

	ELSE
		IF tyP0200OpsGen.tyUSCommB.tyHotspotUSBVSMEMA1.bRtCompl = TRUE THEN
			tyP0200OpsGen.tyUSCommB.tyHotspotUSBVSMEMA1.bRtCompl	:= FALSE;

			IF tyP0200OpsGen.tyUSCommB.tyHotspotUSBVSMEMA1.bValue = TRUE THEN
				bVSMEMAUSBEn	:= TRUE;

				fUIInRtStatOff(ADR(tyP0200OpsGen.tyUSBVSMEMA1.tyLyr.uiRtStat));
				fUIInRtStatHide(ADR(tyP0200OpsGen.tyUSBVSMEMA.tyLyr.uiRtStat));
			ELSE
				tyP0200OpsGen.tyUSBVSMEMA.tyBtnNom.bValue	:= FALSE;
				tyP0200OpsGen.tyUSBVSMEMA.tyBtnStat.bValue	:= FALSE;
				tyP0200OpsGen.tyUSBVSMEMA.tyBtnDual.bValue	:= FALSE;

				bVSMEMAUSBEn	:= FALSE;

				fUIInRtStatHide(ADR(tyP0200OpsGen.tyUSBVSMEMA.tyLyr.uiRtStat));
				fUIInRtStatHide(ADR(tyP0200OpsGen.tyUSBVSMEMA1.tyLyr.uiRtStat));
			END_IF

		END_IF

	END_IF

	//Control

	IF p_tyNtParamCurr.bUIConvDirRL = FALSE THEN

		IF tyP0200OpsGen.tyUSBVSMEMA.tyBtnDual.bRtCompl = TRUE THEN
			tyP0200OpsGen.tyUSBVSMEMA.tyBtnDual.bRtCompl	:= FALSE;

			IF tyP0200OpsGen.tyUSBVSMEMA.tyBtnDual.bValue = TRUE THEN
				tyP0200OpsGen.tyUSBVSMEMA.tyBtnNom.bValue	:= TRUE;
				tyP0200OpsGen.tyUSBVSMEMA.tyBtnStat.bValue	:= TRUE;
			ELSE
				tyP0200OpsGen.tyUSBVSMEMA.tyBtnNom.bValue	:= FALSE;
				tyP0200OpsGen.tyUSBVSMEMA.tyBtnStat.bValue	:= FALSE;
			END_IF

		ELSIF tyP0200OpsGen.tyUSBVSMEMA.tyBtnNom.bRtCompl = TRUE THEN
			tyP0200OpsGen.tyUSBVSMEMA.tyBtnNom.bRtCompl	:= FALSE;

			IF tyP0200OpsGen.tyUSBVSMEMA.tyBtnNom.bValue = TRUE THEN
				IF tyP0200OpsGen.tyUSBVSMEMA.tyBtnStat.bValue =  TRUE THEN
					tyP0200OpsGen.tyUSBVSMEMA.tyBtnDual.bValue	:= TRUE;
				END_IF
			ELSE
				tyP0200OpsGen.tyUSBVSMEMA.tyBtnDual.bValue	:= FALSE;
			END_IF

		ELSIF tyP0200OpsGen.tyUSBVSMEMA.tyBtnStat.bRtCompl = TRUE THEN
			tyP0200OpsGen.tyUSBVSMEMA.tyBtnStat.bRtCompl	:= FALSE;

			IF tyP0200OpsGen.tyUSBVSMEMA.tyBtnStat.bValue = TRUE THEN
				IF tyP0200OpsGen.tyUSBVSMEMA.tyBtnNom.bValue =  TRUE THEN
					tyP0200OpsGen.tyUSBVSMEMA.tyBtnDual.bValue	:= TRUE;
				END_IF
			ELSE
				tyP0200OpsGen.tyUSBVSMEMA.tyBtnDual.bValue	:= FALSE;
			END_IF

		END_IF

	ELSE

		IF tyP0200OpsGen.tyUSBVSMEMA1.tyBtnDual.bRtCompl = TRUE THEN
			tyP0200OpsGen.tyUSBVSMEMA1.tyBtnDual.bRtCompl	:= FALSE;

			IF tyP0200OpsGen.tyUSBVSMEMA1.tyBtnDual.bValue = TRUE THEN
				tyP0200OpsGen.tyUSBVSMEMA1.tyBtnNom.bValue	:= TRUE;
				tyP0200OpsGen.tyUSBVSMEMA1.tyBtnStat.bValue	:= TRUE;
			ELSE
				tyP0200OpsGen.tyUSBVSMEMA1.tyBtnNom.bValue	:= FALSE;
				tyP0200OpsGen.tyUSBVSMEMA1.tyBtnStat.bValue	:= FALSE;
			END_IF

		ELSIF tyP0200OpsGen.tyUSBVSMEMA1.tyBtnNom.bRtCompl = TRUE THEN
			tyP0200OpsGen.tyUSBVSMEMA1.tyBtnNom.bRtCompl	:= FALSE;

			IF tyP0200OpsGen.tyUSBVSMEMA1.tyBtnNom.bValue = TRUE THEN
				IF tyP0200OpsGen.tyUSBVSMEMA1.tyBtnStat.bValue =  TRUE THEN
					tyP0200OpsGen.tyUSBVSMEMA1.tyBtnDual.bValue	:= TRUE;
				END_IF
			ELSE
				tyP0200OpsGen.tyUSBVSMEMA1.tyBtnDual.bValue	:= FALSE;
			END_IF

		ELSIF tyP0200OpsGen.tyUSBVSMEMA1.tyBtnStat.bRtCompl = TRUE THEN
			tyP0200OpsGen.tyUSBVSMEMA1.tyBtnStat.bRtCompl	:= FALSE;

			IF tyP0200OpsGen.tyUSBVSMEMA1.tyBtnStat.bValue = TRUE THEN
				IF tyP0200OpsGen.tyUSBVSMEMA1.tyBtnNom.bValue =  TRUE THEN
					tyP0200OpsGen.tyUSBVSMEMA1.tyBtnDual.bValue	:= TRUE;
				END_IF
			ELSE
				tyP0200OpsGen.tyUSBVSMEMA1.tyBtnDual.bValue	:= FALSE;
			END_IF

		END_IF
	END_IF

	//Update
	IF p_tyNtParamCurr.bUIConvDirRL = FALSE THEN
		bVSMEMAUBAB		:= tyP0200OpsGen.tyUSBVSMEMA.tyBtnNom.bValue;
		bVSMEMAUBABStat	:= tyP0200OpsGen.tyUSBVSMEMA.tyBtnStat.bValue;
	ELSE
		bVSMEMAUBAB		:= tyP0200OpsGen.tyUSBVSMEMA1.tyBtnNom.bValue;
		bVSMEMAUBABStat	:= tyP0200OpsGen.tyUSBVSMEMA1.tyBtnStat.bValue;
	END_IF

END_ACTION
```

#### Act_OptP0200RcyMsg.st
```iecst
ACTION Act_OptP0200RcyMsg:

	//Recovery Message
	FOR i := 1 TO c_uiP0200TableSize DO

		IF tyP0200OpsGen.tyOps.a_tyHotspotRcyMsg[i].bRtCompl = TRUE THEN
			tyP0200OpsGen.tyOps.a_tyHotspotRcyMsg[i].bRtCompl	:= FALSE;

			tyP0200OpsGen.tyRcyMsg.tyTxtMsg.udiValueIdx := p_tyAlarmRcyList[i];

			IF tyP0200OpsGen.tyRcyMsg.tyTxtMsg.udiValueIdx <> 0 THEN
				p_tyC0010RcyMsg ACCESS ADR(tyP0200OpsGen.tyRcyMsg);
			ELSE
				p_tyC0010RcyMsg ACCESS ADR(tyP0200OpsGen.tyRcyMsgHide);
			END_IF

		END_IF

	END_FOR

	//Close Recovery Message
	IF tyP0200OpsGen.tyRcyMsg.tyHotspotClose.bRtCompl = TRUE THEN
		tyP0200OpsGen.tyRcyMsg.tyHotspotClose.bRtCompl	:= FALSE;

		p_tyC0010RcyMsg ACCESS ADR(tyP0200OpsGen.tyRcyMsgHide);
	END_IF

END_ACTION
```

#### Act_EntP0201Disp.st
```iecst
ACTION Act_EntP0201Disp:

	//Access Address
	p_tyC0004Navi ACCESS ADR(tyP0201OpsTravLifter.tyNaviBack);

	p_tyC0005Main ACCESS ADR(tyCommon.tyMain);

	p_tyC0007Notif ACCESS ADR(tyCommon.tyNotif);

	p_tyC0008MsgBox ACCESS ADR(tyP0201OpsTravLifter.tyMsgBoxHide);

	p_tyC0009Info ACCESS ADR(tyCommon.tyInfo);

	p_tyC0011RcpPopUp ACCESS ADR(tyP0201OpsTravLifter.tyRcpPopUp);

	p_tyP0201OpsTravLif ACCESS ADR(tyP0201OpsTravLifter.tyOps);
	p_tyP0201TravLifIOMonitor ACCESS ADR(tyP0201OpsTravLifter.tyIOMonitor);
	p_tyP0201TravLifIOMonitor1 ACCESS ADR (tyP0201OpsTravLifter.tyIOMonitor1);
	p_tyP0201TravLifBypsInitConv ACCESS ADR(tyP0201OpsTravLifter.tyBypsInitConv);
	p_tyP0201Param ACCESS ADR(tyP0201OpsTravLifter.tyParam);

	//Hermes 1.3
	p_tyE0001OpsQueryBoardInfo ACCESS ADR(tyP0201OpsTravLifter.tyQueryBoardInfo);//new for Hermes 1.3
	p_tyE0002OpsCurrWorkOrder ACCESS ADR(tyP0201OpsTravLifter.tyCurrWorkOrderInfo);//new for Hermes 1.3
	p_tyE0003OpsQueryWorkOrder ACCESS ADR(tyP0201OpsTravLifter.tyQueryWorkOrderInfo);//new for Hermes 1.3
	p_tyE0004OpsBarcodeScanner ACCESS ADR(tyP0201OpsTravLifter.tyBarcodeScanner);//new for Hermes 1.3

	//Display
	fUIInRtStatHide(ADR(tyP0201OpsTravLifter.tyIOMonitor.tyLyr.uiRtStat));
	fUIInRtStatHide(ADR(tyP0201OpsTravLifter.tyParam.tyLyr.uiRtStat));

	tyP0201OpsTravLifter.tyOps.tyBtnChgParam.uiRtStat.0	:= NOT(p_tyMcParamCurr.bChgParamEn);

	tyP0201OpsTravLifter.tyParam.tyNumMaxSlt.diValueMax	:= p_tyMagRcpCurrRcp.diTtlSlt;

	//AutoRcp
	IF (p_bMcParamAutoRcpDisable) THEN
		fUIInRtStatOff(ADR(tyP0201OpsTravLifter.tyOps.tyNumPitch.uiRtStat));
		fUIInRtStatOff(ADR(tyP0201OpsTravLifter.tyOps.tyNumMinSltRange.uiRtStat));
		fUIInRtStatOff(ADR(tyP0201OpsTravLifter.tyOps.tyNumMaxSltRange.uiRtStat));
	ELSE
		IF p_tyNtParamCurr.eAutoRcpPrecededBy =  PrecededBySelf THEN
			fUIInRtStatHide(ADR(tyP0201OpsTravLifter.tyOps.tyNumPitch.uiRtStat));
			fUIInRtStatHide(ADR(tyP0201OpsTravLifter.tyOps.tyNumMinSltRange.uiRtStat));
			fUIInRtStatHide(ADR(tyP0201OpsTravLifter.tyOps.tyNumMaxSltRange.uiRtStat));
		ELSIF p_tyNtParamCurr.eAutoRcpPrecededBy =  PrecededByF1 THEN
			fUIInRtStatOff(ADR(tyP0201OpsTravLifter.tyOps.tyNumPitch.uiRtStat));
			fUIInRtStatOff(ADR(tyP0201OpsTravLifter.tyOps.tyNumMinSltRange.uiRtStat));
			fUIInRtStatOff(ADR(tyP0201OpsTravLifter.tyOps.tyNumMaxSltRange.uiRtStat));
		END_IF
	END_IF

END_ACTION
```

#### Act_OptP0201Navi.st
```iecst
ACTION Act_OptP0201Navi:

	IF tyP0201OpsTravLifter.tyNaviBack.tyBtnBack.bRtCompl = TRUE THEN
		tyP0201OpsTravLifter.tyNaviBack.tyBtnBack.bRtCompl	:= FALSE;
		tyP0201OpsTravLifter.tyNaviBack.tyBtnBack.bValue	:= FALSE;

		eChgPage	:= UIP0200OpsGen;

	END_IF

END_ACTION
```

#### Act_OptP0201UpdtDat.st
```iecst
ACTION Act_OptP0201UpdtDat:

	//Status
	fbMcStatUpdtTm(IN := TRUE);
	IF fbMcStatUpdtTm.Q = TRUE THEN
		fbMcStatUpdtTm(IN := FALSE);

		tyP0201OpsTravLifter.tyOps.tyStringMcStat.sValue	:= p_sOpsTravLifULStepTxt;
	END_IF

	//Width
	IF p_tyNtParamCurr.bAWPrep = TRUE AND p_tyMcParamCurr.bAWDis = FALSE THEN
		tyP0201OpsTravLifter.tyOps.tyNumWidth.diValue		:= p_tyMcParamCurr.diWidthAtHmPosInUM - p_diAWOpenActualPos;
		tyP0201OpsTravLifter.tyOps.tyNumWidth2.diValue		:= p_tyMcParamCurr.diWidthAtHmPosInUM - p_diAWOpenActualPos;
	ELSE
		tyP0201OpsTravLifter.tyOps.tyNumWidth.diValue		:= p_tyProdRcpCurrRcp1.diWidthInUM;
		tyP0201OpsTravLifter.tyOps.tyNumWidth2.diValue		:= p_tyProdRcpCurrRcp1.diWidthInUM2;
	END_IF

	//Program Info
	tyP0201OpsTravLifter.tyOps.tyNumMtrPshrExtSpd.diValue	:= p_tyProdRcpCurrRcp1.diMtrPshrExtSpd;
	tyP0201OpsTravLifter.tyOps.tyNumMtrPshrExtTorq.diValue	:= p_tyProdRcpCurrRcp1.diMtrPshrExtTorq;
	tyP0201OpsTravLifter.tyOps.tyNumPshrOffset.diValue		:= p_tyProdRcpCurrRcp1.diPshrOffset;
	IF p_bMcParamAutoRcpDisable OR p_tyNtParamCurr.eAutoRcpPrecededBy =  PrecededByF1 THEN
		tyP0201OpsTravLifter.tyOps.tyTxtMod.usiValueIdx			:= p_tyProdRcpCurrRcp1.usiMcMod;
		tyP0201OpsTravLifter.tyOps.tyStringProdNm.sValue		:= p_tyProdRcpCurrRcp1.sRcpNm;
		tyP0201OpsTravLifter.tyOps.tyBtnToptoBtm.bValue			:= p_tyProdRcpCurrRcp1.bTopToBtm;
		tyP0201OpsTravLifter.tyOps.tyNumMinSltRange.diValue		:= p_tyProdRcpCurrRcp1.diMinSltValue;
		tyP0201OpsTravLifter.tyOps.tyNumMaxSltRange.diValue		:= p_tyProdRcpCurrRcp1.diMaxSltValue;
		tyP0201OpsTravLifter.tyOps.tyNumPitch.diValue			:= p_tyProdRcpCurrRcp1.diPitch;
	ELSE  //FALSE AutoRcp Mode and eAutoRcpPrecededBy = self
		tyP0201OpsTravLifter.tyOps.tyStringProdNm.sValue		:= pa_tyAutoRcpBrdProps[1].sProductTypeId;
		tyP0201OpsTravLifter.tyOps.tyTxtMod.usiValueIdx			:= p_tyProdRcpCurrRcp0.usiMcMod;
		tyP0201OpsTravLifter.tyOps.tyBtnToptoBtm.bValue			:= p_tyProdRcpCurrRcp0.bTopToBtm;
		tyP0201OpsTravLifter.tyOps.tyNumMtrPshrExtSpd.diValue	:= p_tyProdRcpCurrRcp0.diMtrPshrExtSpd;
		tyP0201OpsTravLifter.tyOps.tyNumMtrPshrExtTorq.diValue	:= p_tyProdRcpCurrRcp0.diMtrPshrExtTorq;
		tyP0201OpsTravLifter.tyOps.tyNumPshrOffset.diValue		:= p_tyProdRcpCurrRcp0.diPshrOffset;
	END_IF

	//PCB Status
	IF p_bPshrConvHvBrd = TRUE THEN
		IF p_bPshrConvGdBrd = TRUE THEN
			tyP0201OpsTravLifter.tyOps.tyBitmapPCB.usiValueIdx	:= 1;
		ELSE
			tyP0201OpsTravLifter.tyOps.tyBitmapPCB.usiValueIdx	:= 2;
		END_IF
	ELSE
		tyP0201OpsTravLifter.tyOps.tyBitmapPCB.usiValueIdx	:= 0;
	END_IF

	//Product Recipe 254
	tyP0201OpsTravLifter.tyOps.tyHotspotShowLRcp.uiRtStat.0 := NOT(tyP0201OpsTravLifter.tyOps.tyStringProdNm.sValue <> '');

	IF tyP0201OpsTravLifter.tyOps.tyHotspotShowLRcp.bRtCompl = TRUE THEN
		tyP0201OpsTravLifter.tyOps.tyHotspotShowLRcp.bRtCompl := FALSE;

		fUIInRtStatOff(ADR(tyP0201OpsTravLifter.tyRcpPopUp.tyLyr.uiRtStat));

		tyP0201OpsTravLifter.tyRcpPopUp.tyStringInfo.sValue  := p_tyProdRcpCurrRcp1.sRcpNm;

	ELSIF tyP0201OpsTravLifter.tyRcpPopUp.tyHotspotClose.bRtCompl = TRUE THEN
		tyP0201OpsTravLifter.tyRcpPopUp.tyHotspotClose.bRtCompl := FALSE;

		fUIInRtStatHide(ADR(tyP0201OpsTravLifter.tyRcpPopUp.tyLyr.uiRtStat));
	END_IF

END_ACTION
```

#### Act_OptP0201IOMonitor.st
```iecst
ACTION Act_OptP0201IOMonitor:

	IF tyP0201OpsTravLifter.tyOps.tyHotspotIOMonitor.bRtCompl = TRUE THEN
		tyP0201OpsTravLifter.tyOps.tyHotspotIOMonitor.bRtCompl	:= FALSE;

		fUIInRtStatOff(ADR(tyP0201OpsTravLifter.tyIOMonitor.tyLyr.uiRtStat));

		p_tyC0004Navi ACCESS ADR(tyP0201OpsTravLifter.tyNaviHide);

	ELSIF tyP0201OpsTravLifter.tyIOMonitor.tyHotspotClose.bRtCompl = TRUE THEN
		tyP0201OpsTravLifter.tyIOMonitor.tyHotspotClose.bRtCompl	:= FALSE;
		fUIInRtStatHide(ADR(tyP0201OpsTravLifter.tyIOMonitor.tyLyr.uiRtStat));

		IF bUITravLifShowIOMonitor2 THEN
			fUIInRtStatOff(ADR(tyP0201OpsTravLifter.tyIOMonitor1.tyLyr.uiRtStat));
		ELSE
			p_tyC0004Navi ACCESS ADR(tyP0201OpsTravLifter.tyNaviBack);
		END_IF

	ELSIF tyP0201OpsTravLifter.tyIOMonitor1.tyHotspotClose.bRtCompl = TRUE THEN
		tyP0201OpsTravLifter.tyIOMonitor1.tyHotspotClose.bRtCompl	:= FALSE;

		fUIInRtStatHide(ADR(tyP0201OpsTravLifter.tyIOMonitor1.tyLyr.uiRtStat));

		p_tyC0004Navi ACCESS ADR(tyP0201OpsTravLifter.tyNaviBack);
	END_IF

	IF tyP0201OpsTravLifter.tyIOMonitor.tyLyr.uiRtStat.0 = FALSE THEN

		//Digital Input
		tyP0201OpsTravLifter.tyIOMonitor.tyBtnSafetyRlySig.bValue			:= p_tyDI.bSafetyRlySig;
		tyP0201OpsTravLifter.tyIOMonitor.tyBtnEStop.bValue					:= p_tyDI.bEStopSig;
		tyP0201OpsTravLifter.tyIOMonitor.tyBtnCoverSWSig.bValue				:= p_tyDI.bCoverSWSig;
		tyP0201OpsTravLifter.tyIOMonitor.tyBtnUBAA.bValue					:= p_tyDI.bUBAA;
		tyP0201OpsTravLifter.tyIOMonitor.tyBtnUBAB.bValue					:= p_tyDI.bUBAB;
		tyP0201OpsTravLifter.tyIOMonitor.tyBtnUBAAStat.bValue				:= p_tyDI.bUBAAStat;
		tyP0201OpsTravLifter.tyIOMonitor.tyBtnUBABStat.bValue				:= p_tyDI.bUBABStat;
		tyP0201OpsTravLifter.tyIOMonitor.tyBtnPshrExtRS.bValue				:= p_tyDI.bPusherExtRS;
		tyP0201OpsTravLifter.tyIOMonitor.tyBtnPshrRetRS.bValue				:= p_tyDI.bPusherRetRS;
		tyP0201OpsTravLifter.tyIOMonitor.tyBtnConvLftSen.bValue				:= p_tyDI.bConvLftSen;
		tyP0201OpsTravLifter.tyIOMonitor.tyBtnConvMidSen.bValue				:= p_tyDI.bConvMidSen;
		tyP0201OpsTravLifter.tyIOMonitor.tyBtnConvRgtSen.bValue				:= p_tyDI.bConvRgtSen;
		tyP0201OpsTravLifter.tyIOMonitor.tyBtnConvClrSen.bValue				:= p_tyDI.bConvClrSen;
		tyP0201OpsTravLifter.tyIOMonitor.tyBtnOvenInfeedSigA.bValue			:= p_tyDI.bOvenInfeedSigA;
		tyP0201OpsTravLifter.tyIOMonitor.tyBtnOvenInfeedSigB.bValue			:= p_tyDI.bOvenInfeedSigB;
		tyP0201OpsTravLifter.tyIOMonitor.tyBtnLifterTmBeltSen.bValue		:= p_tyDI.bLifterTimingBeltSen;
		tyP0201OpsTravLifter.tyIOMonitor.tyBtnInletShutterOpenSen.bValue	:= p_tyDI.bInShutterOpenRS;
		tyP0201OpsTravLifter.tyIOMonitor.tyBtnInletShutterCloseSen.bValue	:= p_tyDI.bInShutterCloseRS;
		tyP0201OpsTravLifter.tyIOMonitor.tyBtnOutletShutterOpenSen.bValue	:= p_tyDI.bOutShutterOpenRS;
		tyP0201OpsTravLifter.tyIOMonitor.tyBtnOutletShutterCloseSen.bValue	:= p_tyDI.bOutShutterCloseRS;
		tyP0201OpsTravLifter.tyIOMonitor.tyBtnOutletShutterOpenSen2.bValue	:= p_tyDI.bOutShutterOpenRS2;
		tyP0201OpsTravLifter.tyIOMonitor.tyBtnOutletShutterCloseSen2.bValue	:= p_tyDI.bOutShutterCloseRS2;
		tyP0201OpsTravLifter.tyIOMonitor.tyBtnOutletShutterOpenSen3.bValue	:= p_tyDI.bOutShutterOpenRS3;
		tyP0201OpsTravLifter.tyIOMonitor.tyBtnOutletShutterCloseSen3.bValue	:= p_tyDI.bOutShutterCloseRS3;
		tyP0201OpsTravLifter.tyIOMonitor.tyBtnAntiJamSen.bValue				:= p_tyDI.bPshrAntiJam;
		tyP0201OpsTravLifter.tyIOMonitor.tyBtnInletStopperASensor.bValue	:= p_tyDI.bInletStopperASen;

		//Digital Output
		tyP0201OpsTravLifter.tyIOMonitor.tyBtnSafetyRlyRst.bValue			:= p_tyDO.bSafetyRlyRst;
		tyP0201OpsTravLifter.tyIOMonitor.tyBtnTLGreen.bValue				:= p_tyDO.bTLGreen;
		tyP0201OpsTravLifter.tyIOMonitor.tyBtnTLAmber.bValue				:= p_tyDO.bTLAmber;
		tyP0201OpsTravLifter.tyIOMonitor.tyBtnTLRed.bValue					:= p_tyDO.bTLRed;
		tyP0201OpsTravLifter.tyIOMonitor.tyBtnBuzzer.bValue					:= p_tyDO.bBuzzer;
		tyP0201OpsTravLifter.tyIOMonitor.tyBtnUSBA.bValue					:= p_tyDO.bUSBA;
		tyP0201OpsTravLifter.tyIOMonitor.tyBtnUSBB.bValue					:= p_tyDO.bUSBB;
		tyP0201OpsTravLifter.tyIOMonitor.tyBtnOvenInfoSigA.bValue			:= p_tyDO.bOvenInfoSigA;
		tyP0201OpsTravLifter.tyIOMonitor.tyBtnOvenInfoSigB.bValue			:= p_tyDO.bOvenInfoSigB;
		tyP0201OpsTravLifter.tyIOMonitor.tyBtnPshrExtCtrl.bValue			:= p_tyDO.bPusherExtCtrl;
		tyP0201OpsTravLifter.tyIOMonitor.tyBtnStopperUnBlkCtrlA.bValue		:= p_tyDO.bStopperUnBlkCtrlA;
		tyP0201OpsTravLifter.tyIOMonitor.tyBtnStopperUnBlkCtrlB.bValue		:= p_tyDO.bStopperUnBlkCtrlB;
		tyP0201OpsTravLifter.tyIOMonitor.tyBtnInShutterOpenCtrl.bValue		:= p_tyDO.bInShutterOpenCtrl;
		tyP0201OpsTravLifter.tyIOMonitor.tyBtnInShutterCloseCtrl.bValue		:= p_tyDO.bInShutterCloseCtrl;
		tyP0201OpsTravLifter.tyIOMonitor.tyBtnOutShutterOpenCtrl.bValue		:= p_tyDO.bOutShutterOpenCtrl;
		tyP0201OpsTravLifter.tyIOMonitor.tyBtnOutShutterCloseCtrl.bValue	:= p_tyDO.bOutShutterCloseCtrl;
		tyP0201OpsTravLifter.tyIOMonitor.tyBtnOutShutterOpenCtrl2.bValue	:= p_tyDO.bOutShutterOpenCtrl2;
		tyP0201OpsTravLifter.tyIOMonitor.tyBtnOutShutterCloseCtrl2.bValue	:= p_tyDO.bOutShutterCloseCtrl2;
		tyP0201OpsTravLifter.tyIOMonitor.tyBtnOutShutterOpenCtrl3.bValue	:= p_tyDO.bOutShutterOpenCtrl3;
		tyP0201OpsTravLifter.tyIOMonitor.tyBtnOutShutterCloseCtrl3.bValue	:= p_tyDO.bOutShutterCloseCtrl3;
		tyP0201OpsTravLifter.tyIOMonitor.tyBtnPshrMtrOn.bValue				:= p_tyDO.bPusherConvMtrOn;

	ELSIF tyP0201OpsTravLifter.tyIOMonitor1.tyLyr.uiRtStat.0 = FALSE THEN
		tyP0201OpsTravLifter.tyIOMonitor1.tyBtnScannerComplSig.bValue		:= p_tyDI.diScanComplSig;
		tyP0201OpsTravLifter.tyIOMonitor1.tyBtnPCBPresentSen.bValue			:= p_tyDI.diPCBScanSen;

		tyP0201OpsTravLifter.tyIOMonitor1.tyBtnTrigScannerSig.bValue		:= p_tyDO.diScanTrigSig;
		tyP0201OpsTravLifter.tyIOMonitor1.tyBtnPCBExitMag1.bValue			:= p_tyDO.diMag1ExitPCB;
		tyP0201OpsTravLifter.tyIOMonitor1.tyBtnPCBExitMag2.bValue			:= p_tyDO.diMag2ExitPCB;
		tyP0201OpsTravLifter.tyIOMonitor1.tyBtnPCBExitMag3.bValue			:= p_tyDO.diMag3ExitPCB;
	END_IF

END_ACTION
```

#### Act_OptP0201ChgParam.st
```iecst
ACTION Act_OptP0201ChgParam:

	tyP0201OpsTravLifter.tyParam.tyNumMinSlt.diValueMax			:= tyP0201OpsTravLifter.tyParam.tyNumMaxSlt.diValue;
	tyP0201OpsTravLifter.tyParam.tyNumMaxSlt.diValueMin			:= tyP0201OpsTravLifter.tyParam.tyNumMinSlt.diValue;
	tyP0201OpsTravLifter.tyParam.tyNumPitch.diValueMax			:= tyP0201OpsTravLifter.tyParam.tyNumMaxSlt.diValue - tyP0201OpsTravLifter.tyParam.tyNumMinSlt.diValue + 1;
	tyP0201OpsTravLifter.tyParam.tyNumPitch.diValueMin			:= 1;
	tyP0201OpsTravLifter.tyOps.tyBtnChgParam.uiRtStat.0			:= NOT(p_tyMcParamCurr.bChgParamEn);

	tyP0201OpsTravLifter.tyParam.tyNumPshrExtSpeed.diValueMin 	:= p_tyNtParamCurr.tyProdRcpMtrPshrExtSpd.diMin;
	tyP0201OpsTravLifter.tyParam.tyNumPshrExtSpeed.diValueMax 	:= p_tyNtParamCurr.tyProdRcpMtrPshrExtSpd.diMax;
	tyP0201OpsTravLifter.tyParam.tyNumPshrExtTorque.diValueMin	:= p_tyNtParamCurr.tyProdRcpMtrPshrExtTorq.diMin;
	tyP0201OpsTravLifter.tyParam.tyNumPshrExtTorque.diValueMax	:= p_tyNtParamCurr.tyProdRcpMtrPshrExtTorq.diMax;
	tyP0201OpsTravLifter.tyParam.tyNumPshrExtSpeed.uiRtStat.0	:= NOT p_tyNtParamCurr.bProjMotorizedPusherPrep;
	tyP0201OpsTravLifter.tyParam.tyNumPshrExtTorque.uiRtStat.0	:= NOT p_tyNtParamCurr.bProjMotorizedPusherPrep;

	IF (tyP0201OpsTravLifter.tyOps.tyNumWidth.diValue) <> 0 THEN
		tyP0201OpsTravLifter.tyParam.tyNumPshrOffset.diValueMin := -(tyP0201OpsTravLifter.tyOps.tyNumWidth.diValue/2 - p_tyMcParamCurr.diAWPusherAtHmPosInUM - IPshrSafeDistanceValue);
		tyP0201OpsTravLifter.tyParam.tyNumPshrOffset.diValueMax := (tyP0201OpsTravLifter.tyOps.tyNumWidth.diValue/2 - p_tyMcParamCurr.diAWPusherAtHmPosInUM - IPshrSafeDistanceValue);
	ELSE
		tyP0201OpsTravLifter.tyParam.tyNumPshrOffset.diValueMin := 0;
		tyP0201OpsTravLifter.tyParam.tyNumPshrOffset.diValueMax := 0;
	END_IF

	//Control
	IF tyP0201OpsTravLifter.tyOps.tyBtnChgParam.bRtCompl = TRUE THEN
		tyP0201OpsTravLifter.tyOps.tyBtnChgParam.bRtCompl	:= FALSE;

		tyProdRcpCurrRcpWr	:= p_tyProdRcpCurrRcp0;

		tyP0201OpsTravLifter.tyParam.tyDrpDnMcMode.usiValueIdx	:= p_tyProdRcpCurrRcp0.usiMcMod;
		tyP0201OpsTravLifter.tyParam.tyNumMinSlt.diValue		:= p_tyProdRcpCurrRcp0.diMinSltValue;
		tyP0201OpsTravLifter.tyParam.tyNumMaxSlt.diValue		:= p_tyProdRcpCurrRcp0.diMaxSltValue;
		tyP0201OpsTravLifter.tyParam.tyNumPitch.diValue			:= p_tyProdRcpCurrRcp0.diPitch;
		tyP0201OpsTravLifter.tyParam.tyBtnToptoBtm.bValue		:= p_tyProdRcpCurrRcp0.bTopToBtm;
		tyP0201OpsTravLifter.tyParam.tyNumPshrExtSpeed.diValue 	:= p_tyProdRcpCurrRcp0.diMtrPshrExtSpd;
		tyP0201OpsTravLifter.tyParam.tyNumPshrExtTorque.diValue	:= p_tyProdRcpCurrRcp0.diMtrPshrExtTorq;
		tyP0201OpsTravLifter.tyParam.tyNumPshrOffset.diValue	:= p_tyProdRcpCurrRcp0.diPshrOffset;

		fUIInRtStatOff(ADR(tyP0201OpsTravLifter.tyParam.tyLyr.uiRtStat));

	END_IF

	tyP0201OpsTravLifter.tyOps.tyBtnChgParam.bValue	:= tyP0201OpsTravLifter.tyParam.tyLyr.uiRtStat.0 = FALSE;

	IF tyP0201OpsTravLifter.tyParam.tyLyr.uiRtStat.0 = FALSE THEN

		IF tyP0201OpsTravLifter.tyParam.tyBtnSave.bRtCompl = TRUE THEN

			tyProdRcpCurrRcpWr.usiMcMod			:= tyP0201OpsTravLifter.tyParam.tyDrpDnMcMode.usiValueIdx;
			tyProdRcpCurrRcpWr.diMinSltValue 	:= tyP0201OpsTravLifter.tyParam.tyNumMinSlt.diValue;
			tyProdRcpCurrRcpWr.diMaxSltValue 	:= tyP0201OpsTravLifter.tyParam.tyNumMaxSlt.diValue;
			tyProdRcpCurrRcpWr.diPitch 			:= tyP0201OpsTravLifter.tyParam.tyNumPitch.diValue;
			tyProdRcpCurrRcpWr.bTopToBtm 		:= tyP0201OpsTravLifter.tyParam.tyBtnToptoBtm.bValue;
			tyProdRcpCurrRcpWr.diMtrPshrExtSpd	:= tyP0201OpsTravLifter.tyParam.tyNumPshrExtSpeed.diValue;
			tyProdRcpCurrRcpWr.diMtrPshrExtTorq	:= tyP0201OpsTravLifter.tyParam.tyNumPshrExtTorque.diValue;
			tyProdRcpCurrRcpWr.diPshrOffset		:= tyP0201OpsTravLifter.tyParam.tyNumPshrOffset.diValue;

			eProdRcpAct	:= ProdRcpActWriteCurrRcpParam;

			IF p_eProdRcpStatus = Done AND p_eProdRcpStat = ProdRcpActWriteCurrRcpParam THEN
				eProdRcpAct	:= ProdRcpActIdle;

				//UIP0400
				tyP0400ProdSel.tyProdSel.tyTxtMcMode.usiValueIdx		:= p_tyProdRcpCurrRcp0.usiMcMod;
				tyP0400ProdSel.tyProdSel.tyNumMinSlt.diValue			:= p_tyProdRcpCurrRcp0.diMinSltValue;
				tyP0400ProdSel.tyProdSel.tyNumMaxSlt.diValue			:= p_tyProdRcpCurrRcp0.diMaxSltValue;
				tyP0400ProdSel.tyProdSel.tyNumPitch.diValue				:= p_tyProdRcpCurrRcp0.diPitch;
				tyP0400ProdSel.tyProdSel.tyBtnToptoBtm.bValue			:= p_tyProdRcpCurrRcp0.bTopToBtm;
				tyP0400ProdSel.tyProdSel.tyNumMtrPshrExtSpd.diValue		:= p_tyProdRcpCurrRcp0.diMtrPshrExtSpd;
				tyP0400ProdSel.tyProdSel.tyNumMtrPshrExtTorq.diValue	:= p_tyProdRcpCurrRcp0.diMtrPshrExtTorq;
				tyP0400ProdSel.tyProdSel.tyNumPshrOffset.diValue		:= p_tyProdRcpCurrRcp0.diPshrOffset;

				tyP0201OpsTravLifter.tyParam.tyBtnSave.bRtCompl	:= FALSE;
				tyP0201OpsTravLifter.tyParam.tyBtnSave.bValue	:= FALSE;

				fUIInRtStatHide(ADR(tyP0201OpsTravLifter.tyParam.tyLyr.uiRtStat));

			ELSIF p_eProdRcpStatus = Error THEN
				p_tyC0008MsgBox ACCESS ADR(tyP0201OpsTravLifter.tyMsgBoxSaveErr);

				IF tyP0201OpsTravLifter.tyMsgBoxSaveErr.tyBtnNo.bRtCompl = TRUE THEN
					tyP0201OpsTravLifter.tyMsgBoxSaveErr.tyBtnNo.bRtCompl	:= FALSE;
					tyP0201OpsTravLifter.tyMsgBoxSaveErr.tyBtnNo.bValue		:= FALSE;

					p_tyC0008MsgBox ACCESS ADR(tyP0201OpsTravLifter.tyMsgBoxHide);

					//Restore Param
					tyProdRcpCurrRcpWr	:= p_tyProdRcpCurrRcp0;

					tyP0201OpsTravLifter.tyParam.tyBtnSave.bRtCompl	:= FALSE;
					tyP0201OpsTravLifter.tyParam.tyBtnSave.bValue	:= FALSE;

					fUIInRtStatHide(ADR(tyP0201OpsTravLifter.tyParam.tyLyr.uiRtStat));

				END_IF

			END_IF

		ELSIF tyP0201OpsTravLifter.tyParam.tyBtnCancel.bRtCompl = TRUE THEN
			tyP0201OpsTravLifter.tyParam.tyBtnCancel.bRtCompl	:= FALSE;
			tyP0201OpsTravLifter.tyParam.tyBtnCancel.bValue		:= FALSE;

			fUIInRtStatHide(ADR(tyP0201OpsTravLifter.tyParam.tyLyr.uiRtStat));

		END_IF

	END_IF

	//Mask
	tyP0201OpsTravLifter.tyOps.tyBtnChgParam.uiMaskRtStat.0	:= p_tyUsrMgmtCurrAccessRgt.bChgParam AND p_bOpsStatusStop;

END_ACTION
```

#### Act_OptP0201QueryBoardInfo.st
```iecst
ACTION Act_OptP0201QueryBoardInfo:

	//Hide or Unhide UI button
	IF p_tyHermesConfiguration.a_tyUSParam[0].bFeatureQueryBoardInfo = TRUE AND p_tyNtParamCurr.bHermesPrep AND p_tyMcParamCurr.eUSCommA = McSetCommModHermes THEN
		fUIInRtStatOff(ADR(tyP0201OpsTravLifter.tyOps.tyBtnQueryBoardInfo.uiRtStat)); //show
	ELSE
		fUIInRtStatHide(ADR(tyP0201OpsTravLifter.tyOps.tyBtnQueryBoardInfo.uiRtStat)); //hide
		tyP0201OpsTravLifter.tyOps.tyBtnQueryBoardInfo.bValue := FALSE;
	END_IF

	//Mask
	IF p_tyNtParamCurr.bHermesScannerPrep = TRUE AND p_tyMcParamCurr.bHermesScannerEn = TRUE THEN
		fUIInRtStatHide(ADR(tyP0201OpsTravLifter.tyQueryBoardInfo.tyBtnBarcodeScanner.uiMaskRtStat)); //hide the mask
	ELSE
		fUIInRtStatOff(ADR(tyP0201OpsTravLifter.tyQueryBoardInfo.tyBtnBarcodeScanner.uiMaskRtStat)); //show the mask
	END_IF

	//Press Query Board Info button, bValue will toggle 0,1,0,1.
	IF tyP0201OpsTravLifter.tyOps.tyBtnQueryBoardInfo.bRtCompl = TRUE THEN
		tyP0201OpsTravLifter.tyOps.tyBtnQueryBoardInfo.bRtCompl := FALSE;
	END_IF

	//Popup
	IF 	EDGEPOS (tyP0201OpsTravLifter.tyOps.tyBtnQueryBoardInfo.bValue = TRUE) THEN
		fUIInRtStatOff(ADR(tyP0201OpsTravLifter.tyQueryBoardInfo.tyLyr.uiRtStat)); //show popup QueryBoardInfo
		fUIInRtStatHide(ADR(tyP0201OpsTravLifter.tyBarcodeScanner.tyLyr.uiRtStat)); //hide popup BCScanner
	END_IF

	IF 	EDGEPOS (tyP0201OpsTravLifter.tyQueryBoardInfo.tyBtnBarcodeScanner.bValue = TRUE) THEN
		fUIInRtStatHide(ADR(tyP0201OpsTravLifter.tyQueryBoardInfo.tyLyr.uiRtStat)); //hide popup QueryBoardInfo
		fUIInRtStatOff(ADR(tyP0201OpsTravLifter.tyBarcodeScanner.tyLyr.uiRtStat)); //show popup BCScanner
		fUIInRtStatHide(ADR(tyP0201OpsTravLifter.tyBarcodeScanner.tyBtnTop.uiMaskRtStat)); //hide Mask Top
		fUIInRtStatOff(ADR(tyP0201OpsTravLifter.tyBarcodeScanner.tyBtnMagazine.uiMaskRtStat)); //Mask Magazine
	END_IF

	//Press OK, set bQueryBoardInfo

	IF	tyP0201OpsTravLifter.tyQueryBoardInfo.tyBtnOk.bRtCompl = TRUE THEN

		fUIInRtStatHide(ADR(tyP0201OpsTravLifter.tyQueryBoardInfo.tyLyr.uiRtStat)); //close popup

	    IF (tyP0201OpsTravLifter.tyQueryBoardInfo.tyStringTopBarcode.sValue <> '') OR (tyP0201OpsTravLifter.tyQueryBoardInfo.tyStringBottomBarcode.sValue <> '') THEN

			bQueryBoardInfo := TRUE;
			tyP0201OpsTravLifter.tyOps.tyBtnQueryBoardInfo.bValue := TRUE;
		ELSE
			bQueryBoardInfo := FALSE;
			tyP0201OpsTravLifter.tyOps.tyBtnQueryBoardInfo.bValue := FALSE;
		END_IF

		tyP0201OpsTravLifter.tyQueryBoardInfo.tyBtnOk.bValue := FALSE;

		tyP0201OpsTravLifter.tyQueryBoardInfo.tyBtnOk.bRtCompl := FALSE;

	END_IF

	//Reset
	IF tyP0201OpsTravLifter.tyOps.tyBtnQueryBoardInfo.bValue = FALSE THEN
		bQueryBoardInfo := FALSE;
	END_IF

    //Press Cancel
	IF	tyP0201OpsTravLifter.tyQueryBoardInfo.tyBtnCancel.bRtCompl = TRUE THEN

		fUIInRtStatHide(ADR(tyP0201OpsTravLifter.tyQueryBoardInfo.tyLyr.uiRtStat)); //hide

		tyP0201OpsTravLifter.tyOps.tyBtnQueryBoardInfo.bValue := FALSE;

		tyP0201OpsTravLifter.tyQueryBoardInfo.tyBtnCancel.bRtCompl := FALSE;
		tyP0201OpsTravLifter.tyQueryBoardInfo.tyBtnCancel.bValue := FALSE;
	END_IF

	//Bitmap
	IF tyP0201OpsTravLifter.tyOps.tyBtnQueryBoardInfo.bValue THEN
		tyP0201OpsTravLifter.tyOps.tyBtnQueryBoardInfo.usiBitmapIdx := 1;
	ELSE
		tyP0201OpsTravLifter.tyOps.tyBtnQueryBoardInfo.usiBitmapIdx := 0;
	END_IF

END_ACTION
```

#### Act_OptP0201CurrWorkOrderInfo.st
```iecst
ACTION Act_OptP0201CurrWorkOrderInfo:

	//Hide or Unhide UI button
	IF p_tyHermesConfiguration.tySvyParam.bFeatureQueryWorkOrderInfo = TRUE AND p_tyNtParamCurr.bHermesSvyPrep AND p_tyMcParamCurr.bHermesSvyEn AND p_tyNtParamCurr.bHermesSvyFirstMcInTheLine THEN
		fUIInRtStatOff(ADR(tyP0201OpsTravLifter.tyOps.tyBtnQueryWorkOrderInfo.uiRtStat)); //show
	ELSE
		fUIInRtStatHide(ADR(tyP0201OpsTravLifter.tyOps.tyBtnQueryWorkOrderInfo.uiRtStat)); //hide
		tyP0201OpsTravLifter.tyOps.tyBtnQueryWorkOrderInfo.bValue := FALSE;
	END_IF

	//Press Query Work Order Info button, bValue will toggle.
	IF tyP0201OpsTravLifter.tyOps.tyBtnQueryWorkOrderInfo.bRtCompl = TRUE THEN
		tyP0201OpsTravLifter.tyOps.tyBtnQueryWorkOrderInfo.bRtCompl := FALSE;
	END_IF

	//Popup
	IF 	EDGEPOS (tyP0201OpsTravLifter.tyOps.tyBtnQueryWorkOrderInfo.bValue = TRUE) THEN
		fUIInRtStatOff(ADR(tyP0201OpsTravLifter.tyCurrWorkOrderInfo.tyLyr.uiRtStat)); //show popup View WorkOrder
		fUIInRtStatHide(ADR(tyP0201OpsTravLifter.tyBarcodeScanner.tyLyr.uiRtStat)); //hide popup BCScanner
		fUIInRtStatHide(ADR(tyP0201OpsTravLifter.tyQueryWorkOrderInfo.tyLyr.uiRtStat)); //hide popup QueryWorkOrder
	END_IF

	//Reset
	IF tyP0201OpsTravLifter.tyOps.tyBtnQueryWorkOrderInfo.bValue = FALSE THEN
		bQueryWorkOrderInfo := FALSE;
	END_IF

	//Press Query button, go page QueryWorkOrderInfo
	IF	tyP0201OpsTravLifter.tyCurrWorkOrderInfo.tyBtnQuery.bRtCompl = TRUE AND p_bSiemensMcModeChgPrep = FALSE THEN //AND bDummy THEN

		fUIInRtStatHide(ADR(tyP0201OpsTravLifter.tyCurrWorkOrderInfo.tyLyr.uiRtStat)); //hide popup View WorkOrder
		fUIInRtStatHide(ADR(tyP0201OpsTravLifter.tyBarcodeScanner.tyLyr.uiRtStat)); //hide popup BCScanner
		fUIInRtStatOff(ADR(tyP0201OpsTravLifter.tyQueryWorkOrderInfo.tyLyr.uiRtStat)); //show popup QueryWorkOrder

//		bQueryWorkOrderInfo := TRUE;                                                                  //ADD
//		tyP0201OpsTravLifter.tyOps.tyBtnQueryWorkOrderInfo.bValue := TRUE;

		tyP0201OpsTravLifter.tyCurrWorkOrderInfo.tyBtnQuery.bValue   := FALSE;
		tyP0201OpsTravLifter.tyCurrWorkOrderInfo.tyBtnQuery.bRtCompl := FALSE;

//	ELSE                                                                                            //ADD
//		bQueryWorkOrderInfo := FALSE;
//		tyP0201OpsTravLifter.tyOps.tyBtnQueryWorkOrderInfo.bValue := FALSE;
	ELSIF tyP0201OpsTravLifter.tyCurrWorkOrderInfo.tyBtnQuery.bRtCompl = TRUE (*AND p_bSiemensMcModeChgPrep*) THEN	        //ADD 2022-0780A
		fUIInRtStatHide(ADR(tyP0201OpsTravLifter.tyCurrWorkOrderInfo.tyLyr.uiRtStat)); //hide popup View WorkOrder
		bQueryWorkOrderInfo := TRUE;

		tyP0201OpsTravLifter.tyCurrWorkOrderInfo.tyBtnQuery.bValue   := FALSE;
		tyP0201OpsTravLifter.tyCurrWorkOrderInfo.tyBtnQuery.bRtCompl := FALSE;
	END_IF

	//Manual Query (not possible Traverser in Loader-Unloader)
//	IF (*p_bSiemensMcModeChgPrep AND*) p_bAllZonesEmpty AND p_bOpsConvWaitForTopUpBrd AND  bBypassCoverSwitch = FALSE AND  bTopUpBrdRdy = FALSE AND p_sWorkOrderId <>''  THEN
//		fUIInRtStatHide(ADR(tyP0201OpsTravLifter.tyCurrWorkOrderInfo.tyBtnQuery.uiRtStat)); //hide
//		fUIInRtStatOff(ADR(tyP0201OpsTravLifter.tyCurrWorkOrderInfo.tyBtnDelete.uiRtStat)); //Show
//	ELSIF (*p_bSiemensMcModeChgPrep AND*) p_bAllZonesEmpty AND p_bOpsConvWaitForTopUpBrd AND bBypassCoverSwitch = FALSE AND  bTopUpBrdRdy = FALSE AND p_sWorkOrderId = '' THEN
//		fUIInRtStatOff(ADR(tyP0201OpsTravLifter.tyCurrWorkOrderInfo.tyBtnQuery.uiRtStat)); //Show
//		fUIInRtStatHide(ADR(tyP0201OpsTravLifter.tyCurrWorkOrderInfo.tyBtnDelete.uiRtStat)); //Hide
//	ELSE
//		fUIInRtStatHide(ADR(tyP0201OpsTravLifter.tyCurrWorkOrderInfo.tyBtnQuery.uiRtStat)); //Show
//		fUIInRtStatHide(ADR(tyP0201OpsTravLifter.tyCurrWorkOrderInfo.tyBtnDelete.uiRtStat)); //Hide
//	END_IF

	//Press Exit
	IF	tyP0201OpsTravLifter.tyCurrWorkOrderInfo.tyBtnExit.bRtCompl = TRUE THEN

		fUIInRtStatHide(ADR(tyP0201OpsTravLifter.tyCurrWorkOrderInfo.tyLyr.uiRtStat)); //hide popup View WorkOrder
		fUIInRtStatHide(ADR(tyP0201OpsTravLifter.tyBarcodeScanner.tyLyr.uiRtStat)); //hide popup BCScanner
		fUIInRtStatHide(ADR(tyP0201OpsTravLifter.tyQueryWorkOrderInfo.tyLyr.uiRtStat)); //hide popup QueryWorkOrder

		tyP0201OpsTravLifter.tyOps.tyBtnQueryWorkOrderInfo.bValue := FALSE;

		tyP0201OpsTravLifter.tyCurrWorkOrderInfo.tyBtnExit.bValue   := FALSE;
		tyP0201OpsTravLifter.tyCurrWorkOrderInfo.tyBtnExit.bRtCompl := FALSE;
	END_IF

	tyP0201OpsTravLifter.tyCurrWorkOrderInfo.tyStringWorkOrder.sValue := p_sWorkOrderId;

	//Press Delete, prompt confirm to delete
	IF	tyP0201OpsTravLifter.tyCurrWorkOrderInfo.tyBtnDelete.bRtCompl = TRUE THEN
		p_tyC0008MsgBox ACCESS ADR(tyP0201OpsTravLifter.tyMsgBoxAskDelete);

		IF tyP0201OpsTravLifter.tyMsgBoxAskDelete.tyBtnYes.bRtCompl THEN
		   tyP0201OpsTravLifter.tyMsgBoxAskDelete.tyBtnYes.bRtCompl := FALSE;
			bDeleteWorkOrder := TRUE;
			tyP0201OpsTravLifter.tyCurrWorkOrderInfo.tyBtnDelete.bValue := FALSE;
			tyP0201OpsTravLifter.tyCurrWorkOrderInfo.tyBtnDelete.bRtCompl := FALSE;
			p_tyC0008MsgBox ACCESS ADR(tyP0201OpsTravLifter.tyMsgBoxHide);
			tyP0201OpsTravLifter.tyMsgBoxAskDelete.tyBtnYes.bValue := FALSE;

		ELSIF tyP0201OpsTravLifter.tyMsgBoxAskDelete.tyBtnNo.bRtCompl THEN
			tyP0201OpsTravLifter.tyMsgBoxAskDelete.tyBtnNo.bRtCompl := FALSE;

			bDeleteWorkOrder := FALSE;
			tyP0201OpsTravLifter.tyCurrWorkOrderInfo.tyBtnDelete.bValue := FALSE;
			tyP0201OpsTravLifter.tyCurrWorkOrderInfo.tyBtnDelete.bRtCompl := FALSE;
			p_tyC0008MsgBox ACCESS ADR(tyP0201OpsTravLifter.tyMsgBoxHide);
			tyP0201OpsTravLifter.tyMsgBoxAskDelete.tyBtnNo.bValue := FALSE;
		END_IF

	END_IF

	//Bitmap
	IF tyP0201OpsTravLifter.tyOps.tyBtnQueryWorkOrderInfo.bValue THEN
		tyP0201OpsTravLifter.tyOps.tyBtnQueryWorkOrderInfo.usiBitmapIdx := 1;
	ELSE
		tyP0201OpsTravLifter.tyOps.tyBtnQueryWorkOrderInfo.usiBitmapIdx := 0;
	END_IF

END_ACTION
```

#### Act_OptP0201QueryWorkOrderInfo.st
```iecst
ACTION Act_OptP0201QueryWorkOrderInfo:

	//Mask Magazine Barcode / SlotId
	IF p_tyNtParamCurr.bHermesSvyMagTypeMc = FALSE THEN
		fUIInRtStatOff(ADR(tyP0201OpsTravLifter.tyQueryWorkOrderInfo.tyBitmapMask.uiMaskRtStat)); //show the mask
	ELSE
		fUIInRtStatHide(ADR(tyP0201OpsTravLifter.tyQueryWorkOrderInfo.tyBitmapMask.uiMaskRtStat)); //hide the mask
	END_IF

	//Mask Barcode Scanner
	IF p_tyNtParamCurr.bHermesScannerPrep = TRUE AND p_tyMcParamCurr.bHermesScannerEn = TRUE THEN
		fUIInRtStatHide(ADR(tyP0201OpsTravLifter.tyQueryWorkOrderInfo.tyBtnBarcodeScanner.uiMaskRtStat)); //hide the mask
	ELSE
		fUIInRtStatOff(ADR(tyP0201OpsTravLifter.tyQueryWorkOrderInfo.tyBtnBarcodeScanner.uiMaskRtStat)); //show the mask
	END_IF

	IF 	EDGEPOS (tyP0201OpsTravLifter.tyQueryWorkOrderInfo.tyBtnBarcodeScanner.bValue = TRUE) THEN
		fUIInRtStatHide(ADR(tyP0201OpsTravLifter.tyQueryWorkOrderInfo.tyLyr.uiRtStat)); //hide popup QueryBoardInfo
		fUIInRtStatOff(ADR(tyP0201OpsTravLifter.tyBarcodeScanner.tyLyr.uiRtStat)); //show popup BCScanner
		fUIInRtStatHide(ADR(tyP0201OpsTravLifter.tyBarcodeScanner.tyBtnMagazine.uiMaskRtStat)); //hide Mask Magazine
		fUIInRtStatOff(ADR(tyP0201OpsTravLifter.tyBarcodeScanner.tyBtnTop.uiMaskRtStat)); //Mask Top
	END_IF

	//Convert
	iSlotId := DINT_TO_INT(tyP0201OpsTravLifter.tyQueryWorkOrderInfo.tyNumSlotId.diValue);

	//Press OK, set bQueryWorkOrderInfo
	IF	tyP0201OpsTravLifter.tyQueryWorkOrderInfo.tyBtnOk.bRtCompl = TRUE THEN

		fUIInRtStatHide(ADR(tyP0201OpsTravLifter.tyQueryWorkOrderInfo.tyLyr.uiRtStat)); //close popup

		IF (tyP0201OpsTravLifter.tyQueryWorkOrderInfo.tyStringMagazineId.sValue <> '') OR (iSlotId <> 0)
			OR (tyP0201OpsTravLifter.tyQueryWorkOrderInfo.tyStringBarcode.sValue <> '') THEN
			bQueryWorkOrderInfo := TRUE;
			tyP0201OpsTravLifter.tyOps.tyBtnQueryWorkOrderInfo.bValue := TRUE;
		ELSE
			bQueryWorkOrderInfo := FALSE;
			tyP0201OpsTravLifter.tyOps.tyBtnQueryWorkOrderInfo.bValue := FALSE;
		END_IF

		tyP0201OpsTravLifter.tyQueryWorkOrderInfo.tyBtnOk.bValue := FALSE;

		tyP0201OpsTravLifter.tyQueryWorkOrderInfo.tyBtnOk.bRtCompl := FALSE;

	END_IF

	//Press Cancel
	IF	tyP0201OpsTravLifter.tyQueryWorkOrderInfo.tyBtnCancel.bRtCompl = TRUE THEN

		fUIInRtStatHide(ADR(tyP0201OpsTravLifter.tyQueryWorkOrderInfo.tyLyr.uiRtStat)); //hide
		fUIInRtStatOff(ADR(tyP0201OpsTravLifter.tyCurrWorkOrderInfo.tyLyr.uiRtStat)); //hide

		tyP0201OpsTravLifter.tyQueryWorkOrderInfo.tyBtnCancel.bRtCompl := FALSE;
		tyP0201OpsTravLifter.tyQueryWorkOrderInfo.tyBtnCancel.bValue := FALSE;
	END_IF

END_ACTION
```

#### Act_OptP0201BarcodeScanner.st
```iecst
ACTION Act_OptP0201BarcodeScanner:
	 //Reset bValue
	IF tyP0201OpsTravLifter.tyBarcodeScanner.tyBtnTop.bRtCompl = TRUE  THEN
		tyP0201OpsTravLifter.tyBarcodeScanner.tyBtnTop.bRtCompl := FALSE;

		tyP0201OpsTravLifter.tyBarcodeScanner.tyBtnBottom.bValue := FALSE;
		tyP0201OpsTravLifter.tyBarcodeScanner.tyBtnMagazine.bValue := FALSE;
		tyP0201OpsTravLifter.tyBarcodeScanner.tyBtnPCB.bValue := FALSE;

	END_IF

	IF tyP0201OpsTravLifter.tyBarcodeScanner.tyBtnBottom.bRtCompl = TRUE  THEN
		tyP0201OpsTravLifter.tyBarcodeScanner.tyBtnBottom.bRtCompl := FALSE;

		tyP0201OpsTravLifter.tyBarcodeScanner.tyBtnTop.bValue := FALSE;
		tyP0201OpsTravLifter.tyBarcodeScanner.tyBtnMagazine.bValue := FALSE;
		tyP0201OpsTravLifter.tyBarcodeScanner.tyBtnPCB.bValue := FALSE;
	END_IF

	IF tyP0201OpsTravLifter.tyBarcodeScanner.tyBtnMagazine.bRtCompl = TRUE  THEN
		tyP0201OpsTravLifter.tyBarcodeScanner.tyBtnMagazine.bRtCompl := FALSE;

		tyP0201OpsTravLifter.tyBarcodeScanner.tyBtnTop.bValue := FALSE;
		tyP0201OpsTravLifter.tyBarcodeScanner.tyBtnBottom.bValue := FALSE;
		tyP0201OpsTravLifter.tyBarcodeScanner.tyBtnPCB.bValue := FALSE;
	END_IF

	IF tyP0201OpsTravLifter.tyBarcodeScanner.tyBtnPCB.bRtCompl = TRUE  THEN
		tyP0201OpsTravLifter.tyBarcodeScanner.tyBtnPCB.bRtCompl := FALSE;

		tyP0201OpsTravLifter.tyBarcodeScanner.tyBtnTop.bValue := FALSE;
		tyP0201OpsTravLifter.tyBarcodeScanner.tyBtnBottom.bValue := FALSE;
		tyP0201OpsTravLifter.tyBarcodeScanner.tyBtnMagazine.bValue := FALSE;
	END_IF

	//Top Barcode
	IF EDGEPOS (tyP0201OpsTravLifter.tyBarcodeScanner.tyBtnTop.bValue = TRUE) THEN
		tyP0201OpsTravLifter.tyBarcodeScanner.tyStringBarcode.sValue := tyP0201OpsTravLifter.tyBarcodeScanner.tyStringTopBarcodeBK.sValue;
	END_IF

	IF EDGENEG (tyP0201OpsTravLifter.tyBarcodeScanner.tyBtnTop.bValue = TRUE) THEN
		tyP0201OpsTravLifter.tyBarcodeScanner.tyStringTopBarcodeBK.sValue := tyP0201OpsTravLifter.tyBarcodeScanner.tyStringTopBarcode.sValue;
	END_IF

	IF tyP0201OpsTravLifter.tyBarcodeScanner.tyBtnTop.bValue = TRUE AND tyP0201OpsTravLifter.tyBarcodeScanner.tyBtnBottom.bValue = FALSE  THEN
		tyP0201OpsTravLifter.tyBarcodeScanner.tyStringTopBarcode.sValue := tyP0201OpsTravLifter.tyBarcodeScanner.tyStringBarcode.sValue;
	END_IF

	//Bottom Barcode
	IF EDGEPOS (tyP0201OpsTravLifter.tyBarcodeScanner.tyBtnBottom.bValue = TRUE) THEN
		tyP0201OpsTravLifter.tyBarcodeScanner.tyStringBarcode.sValue := tyP0201OpsTravLifter.tyBarcodeScanner.tyStringBottomBarcodeBK.sValue;
	END_IF

	IF EDGENEG (tyP0201OpsTravLifter.tyBarcodeScanner.tyBtnBottom.bValue = TRUE) THEN
		tyP0201OpsTravLifter.tyBarcodeScanner.tyStringBottomBarcodeBK.sValue := tyP0201OpsTravLifter.tyBarcodeScanner.tyStringBottomBarcode.sValue;
	END_IF

	IF tyP0201OpsTravLifter.tyBarcodeScanner.tyBtnBottom.bValue = TRUE AND tyP0201OpsTravLifter.tyBarcodeScanner.tyBtnTop.bValue = FALSE THEN
		tyP0201OpsTravLifter.tyBarcodeScanner.tyStringBottomBarcode.sValue := tyP0201OpsTravLifter.tyBarcodeScanner.tyStringBarcode.sValue;
	END_IF

	//Magazine Barcode
	IF EDGEPOS (tyP0201OpsTravLifter.tyBarcodeScanner.tyBtnMagazine.bValue = TRUE) THEN
		tyP0201OpsTravLifter.tyBarcodeScanner.tyStringBarcode.sValue := tyP0201OpsTravLifter.tyBarcodeScanner.tyStringMagazineBarcodeBK.sValue;
	END_IF

	IF EDGENEG (tyP0201OpsTravLifter.tyBarcodeScanner.tyBtnMagazine.bValue = TRUE) THEN
		tyP0201OpsTravLifter.tyBarcodeScanner.tyStringMagazineBarcodeBK.sValue := tyP0201OpsTravLifter.tyBarcodeScanner.tyStringMagazineBarcode.sValue;
	END_IF

	IF tyP0201OpsTravLifter.tyBarcodeScanner.tyBtnMagazine.bValue = TRUE AND tyP0201OpsTravLifter.tyBarcodeScanner.tyBtnPCB.bValue = FALSE THEN
		tyP0201OpsTravLifter.tyBarcodeScanner.tyStringMagazineBarcode.sValue := tyP0201OpsTravLifter.tyBarcodeScanner.tyStringBarcode.sValue;
	END_IF

	//PCB Barcode
	IF EDGEPOS (tyP0201OpsTravLifter.tyBarcodeScanner.tyBtnPCB.bValue = TRUE) THEN
		tyP0201OpsTravLifter.tyBarcodeScanner.tyStringBarcode.sValue := tyP0201OpsTravLifter.tyBarcodeScanner.tyStringPCBBarcodeBK.sValue;
	END_IF

	IF EDGENEG (tyP0201OpsTravLifter.tyBarcodeScanner.tyBtnPCB.bValue = TRUE) THEN
		tyP0201OpsTravLifter.tyBarcodeScanner.tyStringPCBBarcodeBK.sValue := tyP0201OpsTravLifter.tyBarcodeScanner.tyStringPCBBarcode.sValue;
	END_IF

	IF tyP0201OpsTravLifter.tyBarcodeScanner.tyBtnPCB.bValue = TRUE AND tyP0201OpsTravLifter.tyBarcodeScanner.tyBtnMagazine.bValue = FALSE THEN
		tyP0201OpsTravLifter.tyBarcodeScanner.tyStringPCBBarcode.sValue := tyP0201OpsTravLifter.tyBarcodeScanner.tyStringBarcode.sValue;
	END_IF

	//Reset to dummy
	IF tyP0201OpsTravLifter.tyBarcodeScanner.tyBtnTop.bValue = FALSE AND  tyP0201OpsTravLifter.tyBarcodeScanner.tyBtnBottom.bValue = FALSE AND tyP0201OpsTravLifter.tyBarcodeScanner.tyBtnMagazine.bValue = FALSE AND tyP0201OpsTravLifter.tyBarcodeScanner.tyBtnPCB.bValue = FALSE THEN
		tyP0201OpsTravLifter.tyBarcodeScanner.tyStringBarcode.sValue := '';
	END_IF

	//Press OK
	IF	tyP0201OpsTravLifter.tyBarcodeScanner.tyBtnOk.bRtCompl = TRUE THEN

		fUIInRtStatHide(ADR(tyP0201OpsTravLifter.tyBarcodeScanner.tyLyr.uiRtStat)); //hide
		IF tyP0201OpsTravLifter.tyOps.tyBtnQueryBoardInfo.bValue THEN
			fUIInRtStatOff(ADR(tyP0201OpsTravLifter.tyQueryBoardInfo.tyLyr.uiRtStat)); //show
			tyP0201OpsTravLifter.tyQueryBoardInfo.tyStringTopBarcode.sValue := tyP0201OpsTravLifter.tyBarcodeScanner.tyStringTopBarcode.sValue;
			tyP0201OpsTravLifter.tyQueryBoardInfo.tyStringBottomBarcode.sValue := tyP0201OpsTravLifter.tyBarcodeScanner.tyStringBottomBarcode.sValue;
		ELSIF tyP0201OpsTravLifter.tyOps.tyBtnQueryWorkOrderInfo.bValue THEN
			fUIInRtStatOff(ADR(tyP0201OpsTravLifter.tyQueryWorkOrderInfo.tyLyr.uiRtStat)); //show
			tyP0201OpsTravLifter.tyQueryWorkOrderInfo.tyStringMagazineId.sValue := tyP0201OpsTravLifter.tyBarcodeScanner.tyStringMagazineBarcode.sValue;
			tyP0201OpsTravLifter.tyQueryWorkOrderInfo.tyStringBarcode.sValue := tyP0201OpsTravLifter.tyBarcodeScanner.tyStringPCBBarcode.sValue;
		END_IF

		tyP0201OpsTravLifter.tyQueryBoardInfo.tyBtnBarcodeScanner.bValue := FALSE;
		tyP0201OpsTravLifter.tyQueryWorkOrderInfo.tyBtnBarcodeScanner.bValue := FALSE;

		tyP0201OpsTravLifter.tyBarcodeScanner.tyBtnOk.bRtCompl := FALSE;
		tyP0201OpsTravLifter.tyBarcodeScanner.tyBtnOk.bValue := FALSE;
		tyP0201OpsTravLifter.tyBarcodeScanner.tyBtnTop.bValue := FALSE;
		tyP0201OpsTravLifter.tyBarcodeScanner.tyBtnBottom.bValue := FALSE;
		tyP0201OpsTravLifter.tyBarcodeScanner.tyBtnMagazine.bValue := FALSE;
		tyP0201OpsTravLifter.tyBarcodeScanner.tyBtnPCB.bValue := FALSE;
		tyP0201OpsTravLifter.tyBarcodeScanner.tyStringBarcode.sValue :='';
		tyP0201OpsTravLifter.tyBarcodeScanner.tyStringTopBarcode.sValue :='';
		tyP0201OpsTravLifter.tyBarcodeScanner.tyStringTopBarcodeBK.sValue :='';
		tyP0201OpsTravLifter.tyBarcodeScanner.tyStringBottomBarcode.sValue :='';
		tyP0201OpsTravLifter.tyBarcodeScanner.tyStringBottomBarcodeBK.sValue :='';
		tyP0201OpsTravLifter.tyBarcodeScanner.tyStringMagazineBarcode.sValue :='';
		tyP0201OpsTravLifter.tyBarcodeScanner.tyStringMagazineBarcodeBK.sValue :='';
		tyP0201OpsTravLifter.tyBarcodeScanner.tyStringPCBBarcode.sValue :='';
		tyP0201OpsTravLifter.tyBarcodeScanner.tyStringPCBBarcodeBK.sValue :='';

	END_IF

	//Press Cancel
	IF	tyP0201OpsTravLifter.tyBarcodeScanner.tyBtnCancel.bRtCompl = TRUE THEN

		fUIInRtStatHide(ADR(tyP0201OpsTravLifter.tyBarcodeScanner.tyLyr.uiRtStat)); //hide
		IF tyP0201OpsTravLifter.tyOps.tyBtnQueryBoardInfo.bValue THEN
			fUIInRtStatOff(ADR(tyP0201OpsTravLifter.tyQueryBoardInfo.tyLyr.uiRtStat)); //show
		ELSIF tyP0201OpsTravLifter.tyOps.tyBtnQueryWorkOrderInfo.bValue THEN
			fUIInRtStatOff(ADR(tyP0201OpsTravLifter.tyQueryWorkOrderInfo.tyLyr.uiRtStat)); //show
		END_IF

		tyP0201OpsTravLifter.tyBarcodeScanner.tyStringBarcode.sValue :='';
		tyP0201OpsTravLifter.tyBarcodeScanner.tyStringTopBarcode.sValue :='';
		tyP0201OpsTravLifter.tyBarcodeScanner.tyStringTopBarcodeBK.sValue :='';
		tyP0201OpsTravLifter.tyBarcodeScanner.tyStringBottomBarcode.sValue :='';
		tyP0201OpsTravLifter.tyBarcodeScanner.tyStringBottomBarcodeBK.sValue :='';
		tyP0201OpsTravLifter.tyBarcodeScanner.tyStringMagazineBarcode.sValue :='';
		tyP0201OpsTravLifter.tyBarcodeScanner.tyStringMagazineBarcodeBK.sValue :='';
		tyP0201OpsTravLifter.tyBarcodeScanner.tyStringPCBBarcode.sValue :='';
		tyP0201OpsTravLifter.tyBarcodeScanner.tyStringPCBBarcodeBK.sValue :='';
		tyP0201OpsTravLifter.tyBarcodeScanner.tyBtnTop.bValue := FALSE;
		tyP0201OpsTravLifter.tyBarcodeScanner.tyBtnBottom.bValue := FALSE;
		tyP0201OpsTravLifter.tyBarcodeScanner.tyBtnMagazine.bValue := FALSE;
		tyP0201OpsTravLifter.tyBarcodeScanner.tyBtnPCB.bValue := FALSE;

		tyP0201OpsTravLifter.tyQueryBoardInfo.tyBtnBarcodeScanner.bValue := FALSE;
		tyP0201OpsTravLifter.tyQueryWorkOrderInfo.tyBtnBarcodeScanner.bValue := FALSE;

		tyP0201OpsTravLifter.tyBarcodeScanner.tyBtnCancel.bRtCompl := FALSE;
		tyP0201OpsTravLifter.tyBarcodeScanner.tyBtnCancel.bValue := FALSE;

	END_IF

END_ACTION
```

#### Act_EntP0202Disp.st
```iecst
ACTION Act_EntP0202Disp:

	//Access Address
	p_tyC0004Navi ACCESS ADR(tyP0202OpsMag1.tyNaviBack);

	p_tyC0005Main ACCESS ADR(tyCommon.tyMain);

	p_tyC0007Notif ACCESS ADR(tyCommon.tyNotif);

	p_tyC0008MsgBox ACCESS ADR(tyP0202OpsMag1.tyMsgBoxHide);

	p_tyC0009Info ACCESS ADR(tyCommon.tyInfo);

	p_tyC0011RcpPopUp ACCESS ADR(tyP0202OpsMag1.tyRcpPopUp);

	p_tyP0202Ops ACCESS ADR(tyP0202OpsMag1.tyOps);
	p_tyP0202IOMonitor ACCESS ADR(tyP0202OpsMag1.tyIOMonitor);
	p_tyP0202BypsInitConv ACCESS ADR(tyP0202OpsMag1.tyBypsInitConv);
	p_tyP0202Param ACCESS ADR(tyP0202OpsMag1.tyParam);
	p_tyP0202ChgMagL1 ACCESS ADR(tyP0202OpsMag1.tyChgMag);
	//DataSource.UI.UI.p_tyP0203ChgMagL2.tyLyr.uiRtStat
	//Display
	fUIInRtStatHide(ADR(tyP0202OpsMag1.tyIOMonitor.tyLyr.uiRtStat));
	fUIInRtStatHide(ADR(tyP0202OpsMag1.tyParam.tyLyr.uiRtStat));

	tyP0202OpsMag1.tyOps.tyBtnChgParam.uiRtStat.0	:= NOT(p_tyMcParamCurr.bChgParamEn);

	IF p_tyNtParamCurr.bMagAutoVerifyPrep = FALSE THEN
		tyP0202OpsMag1.tyIOMonitor.tyBtnMag1FixedClmpRS.usiTxtIdx	:= 70;
		tyP0202OpsMag1.tyIOMonitor.tyBtnMag1FixedUnclmpRS.usiTxtIdx:= 70;
//		tyP0202OpsMag1.tyIOMonitor.tyBtnMag1RmtClmpRS.usiTxtIdx	:= 0;
//		tyP0202OpsMag1.tyIOMonitor.tyBtnMag1RmtUnclmpRS.usiTxtIdx:= 0;
		tyP0202OpsMag1.tyIOMonitor.tyBtnMag1FixedClampCtrl.usiTxtIdx:= 34;
//		tyP0202OpsMag1.tyIOMonitor.tyBtnMag1RemoteClampCtrl.usiTxtIdx:= 0;
	ELSE
	//	tyP0202OpsMag1.tyIOMonitor.tyBtnMag1FixedClmpRS.usiTxtIdx	:= 74;
		tyP0202OpsMag1.tyIOMonitor.tyBtnMag1FixedUnclmpRS.usiTxtIdx:= 70;
	//	tyP0202OpsMag1.tyIOMonitor.tyBtnMag1RmtClmpRS.usiTxtIdx	:= 51;
	//	tyP0202OpsMag1.tyIOMonitor.tyBtnMag1RmtUnclmpRS.usiTxtIdx:= 50;
		tyP0202OpsMag1.tyIOMonitor.tyBtnMag1FixedClampCtrl.usiTxtIdx:=34;
	//	tyP0202OpsMag1.tyIOMonitor.tyBtnMag1RemoteClampCtrl.usiTxtIdx:= 19;

	END_IF

	tyP0202OpsMag1.tyParam.tyNumMaxSlt.diValueMax	:= p_tyMagRcpCurrRcp.diTtlSlt;

END_ACTION
```

#### Act_OptP0202Navi.st
```iecst
ACTION Act_OptP0202Navi:

	IF tyP0202OpsMag1.tyNaviBack.tyBtnBack.bRtCompl = TRUE THEN
		tyP0202OpsMag1.tyNaviBack.tyBtnBack.bRtCompl	:= FALSE;
		tyP0202OpsMag1.tyNaviBack.tyBtnBack.bValue		:= FALSE;

		eChgPage	:= UIP0200OpsGen;

	END_IF

END_ACTION
```

#### Act_OptP0202ChgPage.st
```iecst
ACTION Act_OptP0202ChgPage:

	IF tyP0202OpsMag1.tyOps.tyHotspotMagInfo.bRtCompl = TRUE THEN
		tyP0202OpsMag1.tyOps.tyHotspotMagInfo.bRtCompl	:= FALSE;

		eChgPage	:= UIP0800MagInfo;
	END_IF

END_ACTION
```

#### Act_OptP0202UpdtDat.st
```iecst
ACTION Act_OptP0202UpdtDat:

	//Status
	fbMcStatUpdtTm(IN := TRUE);
	IF fbMcStatUpdtTm.Q = TRUE THEN
		fbMcStatUpdtTm(IN := FALSE);

//		IF p_tyNtParamCurr.bProjMag1ConvPrep = FALSE THEN
//			tyP0202OpsMag1.tyOps.tyStringMcStat.sValue	:= p_sOpsMagUL1StepTxt;
//		ELSE
//			tyP0202OpsMag1.tyOps.tyStringMcStat.sValue	:= p_sOpsMagConvUL1StepTxt;
//		END_IF

		IF p_tyNtParamCurr.bProjLifterMagPlatform THEN
			tyP0202OpsMag1.tyOps.tyStringMcStat.sValue		:= p_sOpsLifMagULStepTxt;
		ELSE
			tyP0202OpsMag1.tyOps.tyStringMcStat.sValue	:= p_sOpsMagConvUL1StepTxt;
		END_IF

	END_IF

	//Width
	IF p_tyNtParamCurr.bAWPrep = TRUE AND p_tyMcParamCurr.bAWDis = FALSE THEN
		tyP0202OpsMag1.tyOps.tyNumWidth.diValue		:= p_tyMcParamCurr.diWidthAtHmPosInUM - p_diAWOpenActualPos;
		tyP0202OpsMag1.tyOps.tyNumWidth2.diValue	:= p_tyMcParamCurr.diWidthAtHmPosInUM - p_diAWOpenActualPos;
	ELSE
		tyP0202OpsMag1.tyOps.tyNumWidth.diValue		:= p_tyProdRcpCurrRcp1.diWidthInUM;
		tyP0202OpsMag1.tyOps.tyNumWidth2.diValue		:= p_tyProdRcpCurrRcp1.diWidthInUM2;
	END_IF

	//Program Info
	IF p_bMcParamAutoRcpDisable OR p_bNtParamAutoRcpF1ArbitraryType  THEN
		tyP0202OpsMag1.tyOps.tyTxtMod.usiValueIdx		:= p_tyProdRcpCurrRcp2.usiMcMod; 		//Mode
		tyP0202OpsMag1.tyOps.tyNumMinSltRange.diValue	:= p_tyProdRcpCurrRcp2.diMinSltValue;
		tyP0202OpsMag1.tyOps.tyNumMaxSltRange.diValue	:= p_tyProdRcpCurrRcp2.diMaxSltValue;
		tyP0202OpsMag1.tyOps.tyBtnToptoBtm.bValue		:= p_tyProdRcpCurrRcp2.bTopToBtm;
		tyP0202OpsMag1.tyOps.tyNumPitch.diValue			:= p_tyProdRcpCurrRcp2.diPitch;
		tyP0202OpsMag1.tyOps.tyStringProdNm.sValue		:= p_tyProdRcpCurrRcp2.sRcpNm;
	ELSE  //FALSE AutoRcp Mode
		tyP0202OpsMag1.tyOps.tyTxtMod.usiValueIdx		:= p_tyProdRcpCurrRcp0.usiMcMod; 		//Mode

		tyP0202OpsMag1.tyOps.tyNumMinSltRange.diValue	:= pa_tyMagProps[1].diMinSlt;
		tyP0202OpsMag1.tyOps.tyNumMaxSltRange.diValue	:= pa_tyMagProps[1].diMaxSlt;
		tyP0202OpsMag1.tyOps.tyBtnToptoBtm.bValue		:= p_tyProdRcpCurrRcp0.bTopToBtm;
		tyP0202OpsMag1.tyOps.tyNumPitch.diValue			:= pa_tyMagProps[1].diPitch;
		IF p_tyNtParamCurr.eAutoRcpPrecededBy =  PrecededBySelf THEN
			tyP0202OpsMag1.tyOps.tyStringProdNm.sValue	:= pa_tyAutoRcpBrdProps[1].sProductTypeId;
		ELSIF p_tyNtParamCurr.eAutoRcpPrecededBy =  PrecededByF1 THEN
			tyP0202OpsMag1.tyOps.tyStringProdNm.sValue	:= pa_tyMagProps[1].sRcpNm;
		END_IF
	END_IF
	//Magazine Info
	tyP0202OpsMag1.tyOps.tyStringMagNm.sValue	:= p_tyMagRcpCurrRcp.sRcpNm;

	IF p_bBuffer1MagPresent = TRUE THEN
		IF p_tyNtParamCurr.eCustomerReq = Siemens AND p_iOpsMagConvUL1MESAcptCond <= 0 AND  p_tyMcParamCurr.bMESEn THEN
			tyP0202OpsMag1.tyOps.tyNumMag1AvlQty.diValue	:= 0;
			tyP0202OpsMag1.tyOps.tyNumMag1TtlSlt.diValue	:= 0;
		ELSE
			tyP0202OpsMag1.tyOps.tyNumMag1AvlQty.diValue	:= p_tyBuffer1BffrStat.diTtlBrdCap - (p_tyBuffer1BffrStat.diTtlGdBrd + p_tyBuffer1BffrStat.diTtlBadBrd);
			tyP0202OpsMag1.tyOps.tyNumMag1TtlSlt.diValue	:= p_tyBuffer1BffrStat.diTtlBrdCap;
		END_IF
	ELSE
		tyP0202OpsMag1.tyOps.tyNumMag1AvlQty.diValue	:= 0;
		tyP0202OpsMag1.tyOps.tyNumMag1TtlSlt.diValue	:= 0;
	END_IF

	//Magazine Present States
	IF p_bBuffer1MagPresent = TRUE THEN

		IF p_tyBuffer1BffrStat.bBffrFull = TRUE THEN
			tyP0202OpsMag1.tyOps.tyTxtMag1Stat.usiValueIdx := 2;
			tyP0202OpsMag1.tyOps.tyTxtMag1Stat.usiColor	   := 1;
		ELSIF p_tyBuffer1BffrStat.bBffrMty = TRUE THEN
			tyP0202OpsMag1.tyOps.tyTxtMag1Stat.usiValueIdx := 1;
			tyP0202OpsMag1.tyOps.tyTxtMag1Stat.usiColor	   := 0;
		ELSE
			tyP0202OpsMag1.tyOps.tyTxtMag1Stat.usiValueIdx := 3;
			tyP0202OpsMag1.tyOps.tyTxtMag1Stat.usiColor	   := 0;
		END_IF

	ELSE
		tyP0202OpsMag1.tyOps.tyTxtMag1Stat.usiValueIdx := 0;
		tyP0202OpsMag1.tyOps.tyTxtMag1Stat.usiColor	   := 1;
	END_IF

	//Product Recipe 254
	tyP0202OpsMag1.tyOps.tyHotspotShowLRcp.uiRtStat.0 := NOT(tyP0202OpsMag1.tyOps.tyStringProdNm.sValue <> '');

	IF tyP0202OpsMag1.tyOps.tyHotspotShowLRcp.bRtCompl = TRUE THEN
		tyP0202OpsMag1.tyOps.tyHotspotShowLRcp.bRtCompl := FALSE;

		fUIInRtStatOff(ADR(tyP0202OpsMag1.tyRcpPopUp.tyLyr.uiRtStat));

		tyP0202OpsMag1.tyRcpPopUp.tyStringInfo.sValue  := p_tyProdRcpCurrRcp1.sRcpNm;

	ELSIF tyP0202OpsMag1.tyRcpPopUp.tyHotspotClose.bRtCompl = TRUE THEN
		tyP0202OpsMag1.tyRcpPopUp.tyHotspotClose.bRtCompl := FALSE;

		fUIInRtStatHide(ADR(tyP0202OpsMag1.tyRcpPopUp.tyLyr.uiRtStat));

	END_IF

END_ACTION
```

#### Act_OptP0202IOMonitor.st
```iecst
ACTION Act_OptP0202IOMonitor:

	IF tyP0202OpsMag1.tyOps.tyHotspotIOMonitor.bRtCompl = TRUE THEN
		tyP0202OpsMag1.tyOps.tyHotspotIOMonitor.bRtCompl	:= FALSE;

		fUIInRtStatOff(ADR(tyP0202OpsMag1.tyIOMonitor.tyLyr.uiRtStat));

		p_tyC0004Navi ACCESS ADR(tyP0202OpsMag1.tyNaviHide);

	ELSIF tyP0202OpsMag1.tyIOMonitor.tyHotspotClose.bRtCompl = TRUE THEN
		tyP0202OpsMag1.tyIOMonitor.tyHotspotClose.bRtCompl	:= FALSE;

		fUIInRtStatHide(ADR(tyP0202OpsMag1.tyIOMonitor.tyLyr.uiRtStat));

		p_tyC0004Navi ACCESS ADR(tyP0202OpsMag1.tyNaviBack);

	END_IF

	IF tyP0202OpsMag1.tyIOMonitor.tyLyr.uiRtStat.0 = FALSE THEN

		//Digital Input
		tyP0202OpsMag1.tyIOMonitor.tyBtnSafetyRlySig.bValue				:= p_tyDI.bSafetyRlySig;
		tyP0202OpsMag1.tyIOMonitor.tyBtnEStop.bValue					:= p_tyDI.bEStopSig;
		tyP0202OpsMag1.tyIOMonitor.tyBtnCoverSWSig.bValue				:= p_tyDI.bCoverSWSig;
		tyP0202OpsMag1.tyIOMonitor.tyBtnUBAA.bValue						:= p_tyDI.bUBAA;
		tyP0202OpsMag1.tyIOMonitor.tyBtnUBAB.bValue						:= p_tyDI.bUBAB;
		tyP0202OpsMag1.tyIOMonitor.tyBtnUBAAStat.bValue					:= p_tyDI.bUBAAStat;
		tyP0202OpsMag1.tyIOMonitor.tyBtnUBABStat.bValue					:= p_tyDI.bUBABStat;
		tyP0202OpsMag1.tyIOMonitor.tyBtnOvenInfeedSigA.bValue			:= p_tyDI.bOvenInfeedSigA;
		tyP0202OpsMag1.tyIOMonitor.tyBtnOvenInfeedSigB.bValue			:= p_tyDI.bOvenInfeedSigB;
		tyP0202OpsMag1.tyIOMonitor.tyBtnMag1FixedClmpRS.bValue			:= p_tyDI.bMag1FixedClampRS;
		tyP0202OpsMag1.tyIOMonitor.tyBtnMag1FixedUnclmpRS.bValue		:= p_tyDI.bMag1FixedUnclampRS;
		tyP0202OpsMag1.tyIOMonitor.tyBtnMag1RmtClmpRS.bValue			:= p_tyDI.bMag1RemoteClampRS;
		tyP0202OpsMag1.tyIOMonitor.tyBtnMag1RmtUnclmpRS.bValue			:= p_tyDI.bMag1RemoteUnclampRS;
		tyP0202OpsMag1.tyIOMonitor.tyBtnMag1ConvEntrySen.bValue			:= p_tyDI.bMagConvEntSen1;
		tyP0202OpsMag1.tyIOMonitor.tyBtnMag1PresentSen.bValue			:= p_tyDI.bMagPresentSen1;
		tyP0202OpsMag1.tyIOMonitor.tyBtnMag1AIVInPosSen1.bValue			:= p_tyDI.bMag1AIVInPosSen1;
		tyP0202OpsMag1.tyIOMonitor.tyBtnMag1AIVInPosSen2.bValue			:= p_tyDI.bMag1AIVInPosSen2;
		tyP0202OpsMag1.tyIOMonitor.tyBtnMag1OrientationChkSen1.bValue	:= p_tyDI.bMag1OrientChkSen1;
		tyP0202OpsMag1.tyIOMonitor.tyBtnMag1OrientationChkSen2.bValue	:= p_tyDI.bMag1OrientChkSen2;

		tyP0202OpsMag1.tyIOMonitor.tyBtnSelUnclampRS.bValue				:= p_tyDI.bMag1SelUnClampRS;

		tyP0202OpsMag1.tyIOMonitor.tyBtnCAB717Sen.bValue				:= p_tyDI.bMagConvCAB717MagSen1;
		tyP0202OpsMag1.tyIOMonitor.tyBtnMagSmallSen.bValue				:= p_tyDI.bMagConvSmallMagSen1;
		tyP0202OpsMag1.tyIOMonitor.tyBtnMagLargeSen.bValue				:= p_tyDI.bMagConvLargeMagSen1;
		tyP0202OpsMag1.tyIOMonitor.tyBtnCurtainSen.bValue				:= p_tyDI.bCurtainSen;
		tyP0202OpsMag1.tyIOMonitor.tyBtnCurtainSenPB.bValue				:= p_tyDI.bCurtainSenPB;
		tyP0202OpsMag1.tyIOMonitor.tyBtnMag1DetSen.bValue				:= p_tyDI.bMag1FixedClampSen;

	IF p_tyNtParamCurr.bMagAutoVerifyPrep = TRUE THEN
		tyP0202OpsMag1.tyIOMonitor.tyBtnHeightSen.bValue				:= p_tyDI.bMagConvHeightSen1;
	ELSE
		tyP0202OpsMag1.tyIOMonitor.tyBtnHeightSen.bValue				:= p_tyDI.bHighMagDetSen1;
	END_IF

		//Digital Output
		tyP0202OpsMag1.tyIOMonitor.tyBtnSafetyRlyRst.bValue				:= p_tyDO.bSafetyRlyRst;
		tyP0202OpsMag1.tyIOMonitor.tyBtnTLGreen.bValue					:= p_tyDO.bTLGreen;
		tyP0202OpsMag1.tyIOMonitor.tyBtnTLAmber.bValue					:= p_tyDO.bTLAmber;
		tyP0202OpsMag1.tyIOMonitor.tyBtnTLRed.bValue					:= p_tyDO.bTLRed;
		tyP0202OpsMag1.tyIOMonitor.tyBtnBuzzer.bValue					:= p_tyDO.bBuzzer;
		tyP0202OpsMag1.tyIOMonitor.tyBtnUSBA.bValue						:= p_tyDO.bUSBA;
		tyP0202OpsMag1.tyIOMonitor.tyBtnUSBB.bValue						:= p_tyDO.bUSBB;
		tyP0202OpsMag1.tyIOMonitor.tyBtnOvenInfoSigA.bValue				:= p_tyDO.bOvenInfoSigA;
		tyP0202OpsMag1.tyIOMonitor.tyBtnOvenInfoSigB.bValue				:= p_tyDO.bOvenInfoSigB;
		tyP0202OpsMag1.tyIOMonitor.tyBtnMag1FixedClampCtrl.bValue		:= p_tyDO.bMag1FixedClampCtrl;
		tyP0202OpsMag1.tyIOMonitor.tyBtnMag1RemoteClampCtrl.bValue		:= p_tyDO.bMag1RemoteClampCtrl;
		tyP0202OpsMag1.tyIOMonitor.tyBtnMag1ConvMtrIn.bValue			:= p_tyDO.bMag1ConvMtrIn;
		tyP0202OpsMag1.tyIOMonitor.tyBtnMag1ConvMtrOut.bValue			:= p_tyDO.bMag1ConvMtrOut;
		tyP0202OpsMag1.tyIOMonitor.tyBtnMagSelClampCtrl.bValue			:= p_tyDO.bMag1SelClampCtrl;
		tyP0202OpsMag1.tyIOMonitor.tyBtnMagSelUnClampCtrl.bValue		:= p_tyDO.bMag1SelUnClampCtrl;
		tyP0202OpsMag1.tyIOMonitor.tyBtnCurtainSenPBLED.bValue			:= p_tyDO.bBypCurtainPBLED;
	END_IF

END_ACTION
```

#### Act_OptP0202_P0003AIVDat.st
```iecst
ACTION Act_OptP0202_P0003AIVDat:

	//Show Change Mag Button only in Manual Exchane Mode
	// insert and remove temporaray replace change magazine button
	tyP0202OpsMag1.tyOps.tyBtnChgMag.uiRtStat.0 := (p_tyMcParamCurr.eMagExMode = McSetMagXcAutoMode AND p_tyMcParamCurr.eAGVComProtocol <> McSetAGVCommDisabled OR p_tyNtParamCurr.bProjLifterMagPlatform) (*OR (p_tyNtParamCurr.bProjBtnInsertRmvMag = FALSE)*);
	tyP0202OpsMag1.tyOps.tyBitmapChgMag.uiRtStat.0 := p_tyMcParamCurr.eMagExMode = McSetMagXcAutoMode  AND p_tyMcParamCurr.eAGVComProtocol <> McSetAGVCommDisabled OR p_tyNtParamCurr.bProjLifterMagPlatform (*OR (p_tyNtParamCurr.bProjBtnInsertRmvMag = FALSE)*);

	//LED Wifi
	tyP0202OpsMag1.tyOps.tyBtnAIVWifi.bValue	:= p_bAGVOnline;

	//Change Magazine
	IF p_tyNtParamCurr.bProjBtnInsertRmvMag = TRUE THEN

		IF EDGENEG(p_bOpsStatusRun) THEN
			bNewMag1	:= FALSE;
			tyP0202OpsMag1.tyOps.tyBtnChgMag.bRtLk	:= FALSE;
			tyP0202OpsMag1.tyOps.tyBtnChgMag.bRtCompl	:= FALSE;
			tyP0003MMenu.tyMMenuBtn.tyBtnRlsNewMag1.bRtLk    := FALSE;
			tyP0003MMenu.tyMMenuBtn.tyBtnRlsNewMag1.bRtCompl := FALSE;
			tyP0202OpsMag1.tyOps.tyBtnChgMag.bValue			:= FALSE;
			tyP0003MMenu.tyMMenuBtn.tyBtnRlsNewMag1.bValue	:= FALSE;
		END_IF

		IF tyP0202OpsMag1.tyOps.tyBtnChgMag.bRtCompl = TRUE OR tyP0003MMenu.tyMMenuBtn.tyBtnRlsNewMag1.bRtCompl THEN
			tyP0202OpsMag1.tyOps.tyBtnChgMag.bRtCompl	:= FALSE;
			tyP0003MMenu.tyMMenuBtn.tyBtnRlsNewMag1.bRtCompl := FALSE;
			bNewMag1	:= p_bOpsMagConvUL1NewMagAllw;
			bRlsMag1	:= p_bOpsMagConvUL1RlsMagAllw;
		END_IF

		IF bNewMag1 = TRUE THEN
			tyP0202OpsMag1.tyOps.tyBitmapChgMag.usiValueIdx	:= 1;
			tyP0003MMenu.tyMMenuBtn.tyBtnRlsNewMag1.usiBitmapIdx := 1;
			IF p_tyDI.bMag1FixedUnclampRS = FALSE THEN
				bNewMag1	:= FALSE;
				tyP0202OpsMag1.tyOps.tyBtnChgMag.bValue	:= FALSE;
				tyP0003MMenu.tyMMenuBtn.tyBtnRlsNewMag1.bValue := FALSE;
				tyP0202OpsMag1.tyOps.tyBtnChgMag.bRtLk	:= FALSE;
				tyP0003MMenu.tyMMenuBtn.tyBtnRlsNewMag1.bRtLk:= FALSE;
				tyP0202OpsMag1.tyOps.tyBitmapChgMag.usiValueIdx	:= 0;
				tyP0003MMenu.tyMMenuBtn.tyBtnRlsNewMag1.usiBitmapIdx := 0;
			END_IF

		ELSIF bRlsMag1 = TRUE THEN
			tyP0202OpsMag1.tyOps.tyBitmapChgMag.usiValueIdx	:= 1;
			tyP0003MMenu.tyMMenuBtn.tyBtnRlsNewMag1.usiBitmapIdx := 1;
			IF p_tyNtParamCurr.eCustomerReq = Siemens THEN
				IF p_bOpsMagConvUL1EjectMESStep THEN //(p_bOpsMagConvUL1EjectMESStep AND p_bOpsMagConvUL1EjectMagNotAllw)
					//OR THEN //FOR MES
					bRlsMag1	:= FALSE;
					tyP0202OpsMag1.tyOps.tyBtnChgMag.bValue	:= FALSE;
					tyP0003MMenu.tyMMenuBtn.tyBtnRlsNewMag1.bValue := FALSE;
					tyP0202OpsMag1.tyOps.tyBtnChgMag.bRtLk	:= FALSE;
					tyP0003MMenu.tyMMenuBtn.tyBtnRlsNewMag1.bRtLk:= FALSE;
					tyP0202OpsMag1.tyOps.tyBitmapChgMag.usiValueIdx	:= 0;
					tyP0003MMenu.tyMMenuBtn.tyBtnRlsNewMag1.usiBitmapIdx := 0;
				END_IF
			ELSIF p_tyDI.bMag1FixedUnclampRS = TRUE AND p_tyDI.bMagPresentSen1 = FALSE  THEN //for Siemen testing
				bRlsMag1	:= FALSE;
				tyP0202OpsMag1.tyOps.tyBtnChgMag.bValue	:= FALSE;
				tyP0003MMenu.tyMMenuBtn.tyBtnRlsNewMag1.bValue := FALSE;
				tyP0202OpsMag1.tyOps.tyBtnChgMag.bRtLk	:= FALSE;
				tyP0003MMenu.tyMMenuBtn.tyBtnRlsNewMag1.bRtLk:= FALSE;
				tyP0202OpsMag1.tyOps.tyBitmapChgMag.usiValueIdx	:= 0;
				tyP0003MMenu.tyMMenuBtn.tyBtnRlsNewMag1.usiBitmapIdx := 0;
			END_IF

		ELSIF p_bAlarmErr THEN
			bNewMag1	:= FALSE;
			bRlsMag1	:= FALSE;
			tyP0202OpsMag1.tyOps.tyBtnChgMag.bValue	:= FALSE;
			tyP0003MMenu.tyMMenuBtn.tyBtnRlsNewMag1.bValue := FALSE;
			tyP0202OpsMag1.tyOps.tyBtnChgMag.bRtLk	:= FALSE;
			tyP0003MMenu.tyMMenuBtn.tyBtnRlsNewMag1.bRtLk:= FALSE;
			tyP0202OpsMag1.tyOps.tyBitmapChgMag.usiValueIdx	:= 0;
			tyP0003MMenu.tyMMenuBtn.tyBtnRlsNewMag1.usiBitmapIdx := 0;
		END_IF

		IF p_tyDI.bMagPresentSen1 AND p_tyDI.bMagConvEntSen1 = FALSE THEN
			tyP0202OpsMag1.tyOps.tyBtnChgMag.usiTxtIdx	:= 1;
			tyP0003MMenu.tyMMenuBtn.tyBtnRlsNewMag1.usiTxtIdx := 31;
		ELSE
			tyP0202OpsMag1.tyOps.tyBtnChgMag.usiTxtIdx	:= 0;
			tyP0003MMenu.tyMMenuBtn.tyBtnRlsNewMag1.usiTxtIdx := 6;
		END_IF

		IF (p_bOpsMagConvUL1NewMagAllw AND p_tyBuffer1BffrStat.bBffrMty)
			OR p_bOpsMagConvUL1RlsMagAllw
			OR p_bBufferMagRemoved1
			THEN //AND p_tyDI.bOutShutterCloseRS
			fUIInRtStatHide(ADR(tyP0202OpsMag1.tyOps.tyBtnChgMag.uiMaskRtStat));
			fUIInRtStatHide(ADR(tyP0003MMenu.tyMMenuBtn.tyBtnRlsNewMag1.uiMaskRtStat));
		ELSE
			fUIInRtStatOff(ADR(tyP0202OpsMag1.tyOps.tyBtnChgMag.uiMaskRtStat));
			fUIInRtStatOff(ADR(tyP0003MMenu.tyMMenuBtn.tyBtnRlsNewMag1.uiMaskRtStat));
		END_IF

	END_IF

END_ACTION
```

#### Act_OptP0202ChgParam.st
```iecst
ACTION Act_OptP0202ChgParam:

	tyP0202OpsMag1.tyParam.tyNumMinSlt.diValueMax		:= tyP0202OpsMag1.tyParam.tyNumMaxSlt.diValue;
	tyP0202OpsMag1.tyParam.tyNumMaxSlt.diValueMin		:= tyP0202OpsMag1.tyParam.tyNumMinSlt.diValue;
	tyP0202OpsMag1.tyParam.tyNumPitch.diValueMax		:= tyP0202OpsMag1.tyParam.tyNumMaxSlt.diValue - tyP0202OpsMag1.tyParam.tyNumMinSlt.diValue + 1;
	tyP0202OpsMag1.tyParam.tyNumPitch.diValueMin		:= 1;
	tyP0202OpsMag1.tyOps.tyBtnChgParam.uiRtStat.0	:= NOT(p_tyMcParamCurr.bChgParamEn);

	tyP0202OpsMag1.tyParam.tyNumPshrExtSpeed.diValueMin 	:= p_tyNtParamCurr.tyProdRcpMtrPshrExtSpd.diMin;
	tyP0202OpsMag1.tyParam.tyNumPshrExtSpeed.diValueMax 	:= p_tyNtParamCurr.tyProdRcpMtrPshrExtSpd.diMax;
	tyP0202OpsMag1.tyParam.tyNumPshrExtTorque.diValueMin	:= p_tyNtParamCurr.tyProdRcpMtrPshrExtTorq.diMin;
	tyP0202OpsMag1.tyParam.tyNumPshrExtTorque.diValueMax	:= p_tyNtParamCurr.tyProdRcpMtrPshrExtTorq.diMax;
	tyP0202OpsMag1.tyParam.tyNumPshrExtSpeed.uiRtStat.0		:= NOT p_tyNtParamCurr.bProjMotorizedPusherPrep;
	tyP0202OpsMag1.tyParam.tyNumPshrExtTorque.uiRtStat.0	:= NOT p_tyNtParamCurr.bProjMotorizedPusherPrep;

	IF (tyP0202OpsMag1.tyOps.tyNumWidth.diValue) <> 0 THEN
		tyP0202OpsMag1.tyParam.tyNumPshrOffset.diValueMin := -(tyP0202OpsMag1.tyOps.tyNumWidth.diValue/2 - p_tyMcParamCurr.diAWPusherAtHmPosInUM - IPshrSafeDistanceValue);
		tyP0202OpsMag1.tyParam.tyNumPshrOffset.diValueMax := (tyP0202OpsMag1.tyOps.tyNumWidth.diValue/2 - p_tyMcParamCurr.diAWPusherAtHmPosInUM - IPshrSafeDistanceValue);
	ELSE
		tyP0202OpsMag1.tyParam.tyNumPshrOffset.diValueMin := 0;
		tyP0202OpsMag1.tyParam.tyNumPshrOffset.diValueMax := 0;
	END_IF

	//Control
	IF 	tyP0202OpsMag1.tyOps.tyBtnChgParam.bRtCompl = TRUE THEN
		tyP0202OpsMag1.tyOps.tyBtnChgParam.bRtCompl	:= FALSE;

		tyProdRcpCurrRcpWr	:= p_tyProdRcpCurrRcp0;

		tyP0202OpsMag1.tyParam.tyDrpDnMcMode.usiValueIdx	:= p_tyProdRcpCurrRcp0.usiMcMod;
		tyP0202OpsMag1.tyParam.tyNumMinSlt.diValue			:= p_tyProdRcpCurrRcp0.diMinSltValue;
		tyP0202OpsMag1.tyParam.tyNumMaxSlt.diValue			:= p_tyProdRcpCurrRcp0.diMaxSltValue;
		tyP0202OpsMag1.tyParam.tyNumPitch.diValue			:= p_tyProdRcpCurrRcp0.diPitch;
		tyP0202OpsMag1.tyParam.tyBtnToptoBtm.bValue			:= p_tyProdRcpCurrRcp0.bTopToBtm;
		tyP0202OpsMag1.tyParam.tyNumPshrExtSpeed.diValue 	:= p_tyProdRcpCurrRcp0.diMtrPshrExtSpd;
		tyP0202OpsMag1.tyParam.tyNumPshrExtTorque.diValue	:= p_tyProdRcpCurrRcp0.diMtrPshrExtTorq;
		tyP0202OpsMag1.tyParam.tyNumPshrOffset.diValue		:= p_tyProdRcpCurrRcp0.diPshrOffset;

		fUIInRtStatOff(ADR(tyP0202OpsMag1.tyParam.tyLyr.uiRtStat));

	END_IF

	tyP0202OpsMag1.tyOps.tyBtnChgParam.bValue		:= tyP0202OpsMag1.tyParam.tyLyr.uiRtStat.0 = FALSE;

	IF tyP0202OpsMag1.tyParam.tyLyr.uiRtStat.0 = FALSE THEN

		IF tyP0202OpsMag1.tyParam.tyBtnSave.bRtCompl = TRUE THEN

			tyProdRcpCurrRcpWr.usiMcMod			:= tyP0202OpsMag1.tyParam.tyDrpDnMcMode.usiValueIdx;
			tyProdRcpCurrRcpWr.diMinSltValue	:= tyP0202OpsMag1.tyParam.tyNumMinSlt.diValue;
			tyProdRcpCurrRcpWr.diMaxSltValue 	:= tyP0202OpsMag1.tyParam.tyNumMaxSlt.diValue;
			tyProdRcpCurrRcpWr.diPitch 			:= tyP0202OpsMag1.tyParam.tyNumPitch.diValue;
			tyProdRcpCurrRcpWr.bTopToBtm 		:= tyP0202OpsMag1.tyParam.tyBtnToptoBtm.bValue;
			tyProdRcpCurrRcpWr.diMtrPshrExtSpd	:= tyP0202OpsMag1.tyParam.tyNumPshrExtSpeed.diValue;
			tyProdRcpCurrRcpWr.diMtrPshrExtTorq	:= tyP0202OpsMag1.tyParam.tyNumPshrExtTorque.diValue;
			tyProdRcpCurrRcpWr.diPshrOffset		:= tyP0202OpsMag1.tyParam.tyNumPshrOffset.diValue;

			eProdRcpAct	:= ProdRcpActWriteCurrRcpParam;

			IF p_eProdRcpStatus = Done AND p_eProdRcpStat = ProdRcpActWriteCurrRcpParam THEN
				eProdRcpAct	:= ProdRcpActIdle;

				//UIP0400
				tyP0400ProdSel.tyProdSel.tyTxtMcMode.usiValueIdx		:= p_tyProdRcpCurrRcp0.usiMcMod;
				tyP0400ProdSel.tyProdSel.tyNumMinSlt.diValue			:= p_tyProdRcpCurrRcp0.diMinSltValue;
				tyP0400ProdSel.tyProdSel.tyNumMaxSlt.diValue			:= p_tyProdRcpCurrRcp0.diMaxSltValue;
				tyP0400ProdSel.tyProdSel.tyNumPitch.diValue				:= p_tyProdRcpCurrRcp0.diPitch;
				tyP0400ProdSel.tyProdSel.tyBtnToptoBtm.bValue			:= p_tyProdRcpCurrRcp0.bTopToBtm;
				tyP0400ProdSel.tyProdSel.tyNumMtrPshrExtSpd.diValue		:= p_tyProdRcpCurrRcp0.diMtrPshrExtSpd;
				tyP0400ProdSel.tyProdSel.tyNumMtrPshrExtTorq.diValue	:= p_tyProdRcpCurrRcp0.diMtrPshrExtTorq;
				tyP0400ProdSel.tyProdSel.tyNumPshrOffset.diValue		:= p_tyProdRcpCurrRcp0.diPshrOffset;

				tyP0202OpsMag1.tyParam.tyBtnSave.bRtCompl			:= FALSE;
				tyP0202OpsMag1.tyParam.tyBtnSave.bValue				:= FALSE;

				fUIInRtStatHide(ADR(tyP0202OpsMag1.tyParam.tyLyr.uiRtStat));

			ELSIF p_eProdRcpStatus = Error THEN
				p_tyC0008MsgBox ACCESS ADR(tyP0202OpsMag1.tyMsgBoxSaveErr);

				IF tyP0202OpsMag1.tyMsgBoxSaveErr.tyBtnNo.bRtCompl = TRUE THEN
					tyP0202OpsMag1.tyMsgBoxSaveErr.tyBtnNo.bRtCompl	:= FALSE;
					tyP0202OpsMag1.tyMsgBoxSaveErr.tyBtnNo.bValue	:= FALSE;

					p_tyC0008MsgBox ACCESS ADR(tyP0202OpsMag1.tyMsgBoxHide);

					//Restore Param
					tyProdRcpCurrRcpWr	:= p_tyProdRcpCurrRcp2;

					tyP0202OpsMag1.tyParam.tyBtnSave.bRtCompl		:= FALSE;
					tyP0202OpsMag1.tyParam.tyBtnSave.bValue			:= FALSE;

					fUIInRtStatHide(ADR(tyP0202OpsMag1.tyParam.tyLyr.uiRtStat));

				END_IF

			END_IF

		ELSIF tyP0202OpsMag1.tyParam.tyBtnCancel.bRtCompl = TRUE THEN
			tyP0202OpsMag1.tyParam.tyBtnCancel.bRtCompl				:= FALSE;
			tyP0202OpsMag1.tyParam.tyBtnCancel.bValue				:= FALSE;

			fUIInRtStatHide(ADR(tyP0202OpsMag1.tyParam.tyLyr.uiRtStat));

		END_IF

	END_IF

	//Mask
	tyP0202OpsMag1.tyOps.tyBtnChgParam.uiMaskRtStat.0	:= p_tyUsrMgmtCurrAccessRgt.bChgParam AND p_bOpsStatusStop;

END_ACTION
```
